	Nr_100		:BOOL;// #MText: #HText: #Prio: #BMK:
	Nr_101		:BOOL;// #MText: #HText: #Prio: #BMK:
	Nr_102		:BOOL;// #MText: #HText: #Prio: #BMK:
	Nr_103		:BOOL;// #MText: #HText: #Prio: #BMK:
	Nr_104		:BOOL;// #MText: #HText: #Prio: #BMK:
	Nr_105		:BOOL;// #MText: #HText: #Prio: #BMK:
	Nr_106		:BOOL;// #MText: #HText: #Prio: #BMK:
	Nr_107		:BOOL;// #MText: #HText: #Prio: #BMK:
	Nr_108		:BOOL;// #MText: #HText: #Prio: #BMK:
	Nr_109		:BOOL;// #MText: #HText: #Prio: #BMK:
	Nr_110		:BOOL;// #MText: #HText: #Prio: #BMK:
	Nr_111		:BOOL;// #MText: #HText: #Prio: #BMK:
	Nr_112		:BOOL;// #MText: #HText: #Prio: #BMK:
	Nr_113		:BOOL;// #MText: #HText: #Prio: #BMK:
	Nr_114		:BOOL;// #MText: #HText: #Prio: #BMK:
	Nr_115		:BOOL;// #MText: #HText: #Prio: #BMK:
	Nr_116		:BOOL;// #MText: #HText: #Prio: #BMK:
	Nr_117		:BOOL;// #MText: #HText: #Prio: #BMK:
	Nr_118		:BOOL;// #MText: #HText: #Prio: #BMK:
	Nr_119		:BOOL;// #MText: #HText: #Prio: #BMK:
	Nr_120		:BOOL;// #MText: #HText: #Prio: #BMK:
	Nr_121		:BOOL;// #MText: #HText: #Prio: #BMK:
	Nr_122		:BOOL;// #MText: #HText: #Prio: #BMK:
	Nr_123		:BOOL;// #MText: #HText: #Prio: #BMK:
	Nr_124		:BOOL;// #MText: #HText: #Prio: #BMK:
	Nr_125		:BOOL;// #MText: #HText: #Prio: #BMK:
	Nr_126		:BOOL;// #MText: #HText: #Prio: #BMK:
	Nr_127		:BOOL;// #MText: #HText: #Prio: #BMK:
	Nr_128		:BOOL;// #MText: #HText: #Prio: #BMK:
	Nr_129		:BOOL;// #MText: #HText: #Prio: #BMK:
	Nr_130		:BOOL;// #MText: #HText: #Prio: #BMK:
	Nr_131		:BOOL;// #MText: #HText: #Prio: #BMK:
	Nr_132		:BOOL;// #MText: #HText: #Prio: #BMK:
	Nr_133		:BOOL;// #MText: #HText: #Prio: #BMK:
	Nr_134		:BOOL;// #MText: #HText: #Prio: #BMK:
	Nr_135		:BOOL;// #MText: #HText: #Prio: #BMK:
	Nr_136		:BOOL;// #MText: #HText: #Prio: #BMK:
	Nr_137		:BOOL;// #MText: #HText: #Prio: #BMK:
	Nr_138		:BOOL;// #MText: #HText: #Prio: #BMK:
	Nr_139		:BOOL;// #MText: #HText: #Prio: #BMK:
	Nr_140		:BOOL;// #MText: #HText: #Prio: #BMK:
	Nr_141		:BOOL;// #MText: #HText: #Prio: #BMK:
	Nr_142		:BOOL;// #MText: #HText: #Prio: #BMK:
	Nr_143		:BOOL;// #MText: #HText: #Prio: #BMK:
	Nr_144		:BOOL;// #MText: #HText: #Prio: #BMK:
	Nr_145		:BOOL;// #MText: #HText: #Prio: #BMK:
	Nr_146		:BOOL;// #MText: #HText: #Prio: #BMK:
	Nr_147		:BOOL;// #MText: #HText: #Prio: #BMK:
	Nr_148		:BOOL;// #MText: #HText: #Prio: #BMK:
	Nr_149		:BOOL;// #MText: #HText: #Prio: #BMK:
	Nr_150		:BOOL;// #MText: #HText: #Prio: #BMK:
	Nr_151		:BOOL;// #MText: #HText: #Prio: #BMK:
	Nr_152		:BOOL;// #MText: #HText: #Prio: #BMK:
	Nr_153		:BOOL;// #MText: #HText: #Prio: #BMK:
	Nr_154		:BOOL;// #MText: #HText: #Prio: #BMK:
	Nr_155		:BOOL;// #MText: #HText: #Prio: #BMK:
	Nr_156		:BOOL;// #MText: #HText: #Prio: #BMK:
	Nr_157		:BOOL;// #MText: #HText: #Prio: #BMK:
	Nr_158		:BOOL;// #MText: #HText: #Prio: #BMK:
	Nr_159		:BOOL;// #MText: #HText: #Prio: #BMK:
	Nr_160		:BOOL;// #MText: #HText: #Prio: #BMK:
	Nr_161		:BOOL;// #MText: #HText: #Prio: #BMK:
	Nr_162		:BOOL;// #MText: #HText: #Prio: #BMK:
	Nr_163		:BOOL;// #MText: #HText: #Prio: #BMK:
	Nr_164		:BOOL;// #MText: #HText: #Prio: #BMK:
	Nr_165		:BOOL;// #MText: #HText: #Prio: #BMK:
	Nr_166		:BOOL;// #MText: #HText: #Prio: #BMK:
	Nr_167		:BOOL;// #MText: #HText: #Prio: #BMK:
	Nr_168		:BOOL;// #MText: #HText: #Prio: #BMK:
	Nr_169		:BOOL;// #MText: #HText: #Prio: #BMK:
	Nr_170		:BOOL;// #MText: #HText: #Prio: #BMK:
	Nr_171		:BOOL;// #MText: #HText: #Prio: #BMK:
	Nr_172		:BOOL;// #MText: #HText: #Prio: #BMK:
	Nr_173		:BOOL;// #MText: #HText: #Prio: #BMK:
	Nr_174		:BOOL;// #MText: #HText: #Prio: #BMK:
	Nr_175		:BOOL;// #MText: #HText: #Prio: #BMK:
	Nr_176		:BOOL;// #MText: #HText: #Prio: #BMK:
	Nr_177		:BOOL;// #MText: #HText: #Prio: #BMK:
	Nr_178		:BOOL;// #MText: #HText: #Prio: #BMK:
	Nr_179		:BOOL;// #MText: #HText: #Prio: #BMK:
	Nr_180		:BOOL;// #MText: #HText: #Prio: #BMK:
	Nr_181		:BOOL;// #MText: #HText: #Prio: #BMK:
	Nr_182		:BOOL;// #MText: #HText: #Prio: #BMK:
	Nr_183		:BOOL;// #MText: #HText: #Prio: #BMK:
	Nr_184		:BOOL;// #MText: #HText: #Prio: #BMK:
	Nr_185		:BOOL;// #MText: #HText: #Prio: #BMK:
	Nr_186		:BOOL;// #MText: #HText: #Prio: #BMK:
	Nr_187		:BOOL;// #MText: #HText: #Prio: #BMK:
	Nr_188		:BOOL;// #MText: #HText: #Prio: #BMK:
	Nr_189		:BOOL;// #MText: #HText: #Prio: #BMK:
	Nr_190		:BOOL;// #MText: #HText: #Prio: #BMK:
	Nr_191		:BOOL;// #MText: #HText: #Prio: #BMK:
	Nr_192		:BOOL;// #MText: #HText: #Prio: #BMK:
	Nr_193		:BOOL;// #MText: #HText: #Prio: #BMK:
	Nr_194		:BOOL;// #MText: #HText: #Prio: #BMK:
	Nr_195		:BOOL;// #MText: #HText: #Prio: #BMK:
	Nr_196		:BOOL;// #MText: #HText: #Prio: #BMK:
	Nr_197		:BOOL;// #MText: #HText: #Prio: #BMK:
	Nr_198		:BOOL;// #MText: #HText: #Prio: #BMK:
	Nr_199		:BOOL;// #MText: #HText: #Prio: #BMK:
	
END_STRUCT
END_TYPE

// ---- SRT_Allgemein/0010_Bausteine_mitDuts/DUTs/Meldungen/DUT_Meldungen_5000.TcDUT
TYPE DUT_Meldungen_5000 :
STRUCT
					  // #MText: Achtung ein Fehler #HText: Achtung eine Hilfe #Prio: 1-10 Error 11-20 Warnung 21-30 Info #BMK:	

	Nr_001		:BOOL;// #MText: #HText: #Prio: #BMK:
	Nr_002		:BOOL;// #MText: #HText: #Prio: #BMK: 
	Nr_003		:BOOL;// #MText: #HText: #Prio: #BMK: 
	Nr_004		:BOOL;// #MText: #HText: #Prio: #BMK: 
	Nr_005		:BOOL;// #MText: #HText: #Prio: #BMK: 
	Nr_006		:BOOL;// #MText: #HText: #Prio: #BMK: 
	Nr_007		:BOOL;// #MText: #HText: #Prio: #BMK: 
	Nr_008		:BOOL;// #MText: #HText: #Prio: #BMK: 
	Nr_009		:BOOL;// #MText: #HText: #Prio: #BMK: 
	Nr_010		:BOOL;// #MText: #HText: #Prio: #BMK: 
	Nr_011		:BOOL;// #MText: #HText: #Prio: #BMK: 
	Nr_012		:BOOL;// #MText: #HText: #Prio: #BMK: 
	Nr_013		:BOOL;// #MText: #HText: #Prio: #BMK: 
	Nr_014		:BOOL;// #MText: #HText: #Prio: #BMK: 
	Nr_015		:BOOL;// #MText: #HText: #Prio: #BMK:     
	Nr_016		:BOOL;// #MText: #HText: #Prio: #BMK:
	Nr_017		:BOOL;// #MText: #HText: #Prio: #BMK:     
	Nr_018		:BOOL;// #MText: #HText: #Prio: #BMK:
	Nr_019		:BOOL;// #MText: #HText: #Prio: #BMK:     
	Nr_020		:BOOL;// #MText: #HText: #Prio: #BMK:
	Nr_021		:BOOL;// #MText: #HText: #Prio: #BMK:     
	Nr_022		:BOOL;// #MText: #HText: #Prio: #BMK:     
	Nr_023		:BOOL;// #MText: #HText: #Prio: #BMK:      
	Nr_024		:BOOL;// #MText: #HText: #Prio: #BMK:
	Nr_025		:BOOL;// #MText: #HText: #Prio: #BMK:      
	Nr_026		:BOOL;// #MText: #HText: #Prio: #BMK:
	Nr_027		:BOOL;// #MText: #HText: #Prio: #BMK:      
	Nr_028		:BOOL;// #MText: #HText: #Prio: #BMK:
	Nr_029		:BOOL;// #MText: #HText: #Prio: #BMK:      
	Nr_030		:BOOL;// #MText: #HText: #Prio: #BMK:
	Nr_031		:BOOL;// #MText: #HText: #Prio: #BMK:      
	Nr_032		:BOOL;// #MText: #HText: #Prio: #BMK:
	Nr_033		:BOOL;// #MText: #HText: #Prio: #BMK:      
	Nr_034		:BOOL;// #MText: #HText: #Prio: #BMK:
	Nr_035		:BOOL;// #MText: #HText: #Prio: #BMK:      
	Nr_036		:BOOL;// #MText: #HText: #Prio: #BMK:
	Nr_037		:BOOL;// #MText: #HText: #Prio: #BMK:
	Nr_038		:BOOL;// #MText: #HText: #Prio: #BMK:
	Nr_039		:BOOL;// #MText: #HText: #Prio: #BMK:
	Nr_040		:BOOL;// #MText: #HText: #Prio: #BMK:
	Nr_041		:BOOL;// #MText: #HText: #Prio: #BMK:
	Nr_042		:BOOL;// #MText: #HText: #Prio: #BMK:
	Nr_043		:BOOL;// #MText: #HText: #Prio: #BMK:
	Nr_044		:BOOL;// #MText: #HText: #Prio: #BMK:
	Nr_045		:BOOL;// #MText: #HText: #Prio: #BMK:
	Nr_046		:BOOL;// #MText: #HText: #Prio: #BMK:
	Nr_047		:BOOL;// #MText: #HText: #Prio: #BMK:
	Nr_048		:BOOL;// #MText: #HText: #Prio: #BMK:
	Nr_049		:BOOL;// #MText: #HText: #Prio: #BMK:
	Nr_050		:BOOL;// #MText: #HText: #Prio: #BMK:
	Nr_051		:BOOL;// #MText: #HText: #Prio: #BMK:
	Nr_052		:BOOL;// #MText: #HText: #Prio: #BMK:
	Nr_053		:BOOL;// #MText: #HText: #Prio: #BMK:
	Nr_054		:BOOL;// #MText: #HText: #Prio: #BMK:
	Nr_055		:BOOL;// #MText: #HText: #Prio: #BMK:
	Nr_056		:BOOL;// #MText: #HText: #Prio: #BMK:
	Nr_057		:BOOL;// #MText: #HText: #Prio: #BMK:
	Nr_058		:BOOL;// #MText: #HText: #Prio: #BMK:
	Nr_059		:BOOL;// #MText: #HText: #Prio: #BMK:
	Nr_060		:BOOL;// #MText: #HText: #Prio: #BMK:
	Nr_061		:BOOL;// #MText: #HText: #Prio: #BMK:
	Nr_062		:BOOL;// #MText: #HText: #Prio: #BMK:
	Nr_063		:BOOL;// #MText: #HText: #Prio: #BMK:
	Nr_064		:BOOL;// #MText: #HText: #Prio: #BMK:
	Nr_065		:BOOL;// #MText: #HText: #Prio: #BMK:
	Nr_066		:BOOL;// #MText: #HText: #Prio: #BMK:
	Nr_067		:BOOL;// #MText: #HText: #Prio: #BMK:
	Nr_068		:BOOL;// #MText: #HText: #Prio: #BMK:
	Nr_069		:BOOL;// #MText: #HText: #Prio: #BMK:
	Nr_070		:BOOL;// #MText: #HText: #Prio: #BMK:
	Nr_071		:BOOL;// #MText: #HText: #Prio: #BMK:
	Nr_072		:BOOL;// #MText: #HText: #Prio: #BMK:
	Nr_073		:BOOL;// #MText: #HText: #Prio: #BMK:
	Nr_074		:BOOL;// #MText: #HText: #Prio: #BMK:
	Nr_075		:BOOL;// #MText: #HText: #Prio: #BMK:
	Nr_076		:BOOL;// #MText: #HText: #Prio: #BMK:
	Nr_077		:BOOL;// #MText: #HText: #Prio: #BMK:
	Nr_078		:BOOL;// #MText: #HText: #Prio: #BMK:
	Nr_079		:BOOL;// #MText: #HText: #Prio: #BMK:
	Nr_080		:BOOL;// #MText: #HText: #Prio: #BMK:
	Nr_081		:BOOL;// #MText: #HText: #Prio: #BMK:
	Nr_082		:BOOL;// #MText: #HText: #Prio: #BMK:
	Nr_083		:BOOL;// #MText: #HText: #Prio: #BMK:
	Nr_084		:BOOL;// #MText: #HText: #Prio: #BMK:
	Nr_085		:BOOL;// #MText: #HText: #Prio: #BMK:
	Nr_086		:BOOL;// #MText: #HText: #Prio: #BMK:
	Nr_087		:BOOL;// #MText: #HText: #Prio: #BMK:
	Nr_088		:BOOL;// #MText: #HText: #Prio: #BMK:
	Nr_089		:BOOL;// #MText: #HText: #Prio: #BMK:
	Nr_090		:BOOL;// #MText: #HText: #Prio: #BMK:
	Nr_091		:BOOL;// #MText: #HText: #Prio: #BMK:
	Nr_092		:BOOL;// #MText: #HText: #Prio: #BMK:
	Nr_093		:BOOL;// #MText: #HText: #Prio: #BMK:
	Nr_094		:BOOL;// #MText: #HText: #Prio: #BMK:
	Nr_095		:BOOL;// #MText: #HText: #Prio: #BMK:
	Nr_096		:BOOL;// #MText: #HText: #Prio: #BMK:
	Nr_097		:BOOL;// #MText: #HText: #Prio: #BMK:
	Nr_098		:BOOL;// #MText: #HText: #Prio: #BMK:
	Nr_099		:BOOL;// #MText: #HText: #Prio: #BMK:
	
	Nr_100		:BOOL;// #MText: #HText: #Prio: #BMK:
	Nr_101		:BOOL;// #MText: #HText: #Prio: #BMK:
	Nr_102		:BOOL;// #MText: #HText: #Prio: #BMK:
	Nr_103		:BOOL;// #MText: #HText: #Prio: #BMK:
	Nr_104		:BOOL;// #MText: #HText: #Prio: #BMK:
	Nr_105		:BOOL;// #MText: #HText: #Prio: #BMK:
	Nr_106		:BOOL;// #MText: #HText: #Prio: #BMK:
	Nr_107		:BOOL;// #MText: #HText: #Prio: #BMK:
	Nr_108		:BOOL;// #MText: #HText: #Prio: #BMK:
	Nr_109		:BOOL;// #MText: #HText: #Prio: #BMK:
	Nr_110		:BOOL;// #MText: #HText: #Prio: #BMK:
	Nr_111		:BOOL;// #MText: #HText: #Prio: #BMK:
	Nr_112		:BOOL;// #MText: #HText: #Prio: #BMK:
	Nr_113		:BOOL;// #MText: #HText: #Prio: #BMK:
	Nr_114		:BOOL;// #MText: #HText: #Prio: #BMK:
	Nr_115		:BOOL;// #MText: #HText: #Prio: #BMK:
	Nr_116		:BOOL;// #MText: #HText: #Prio: #BMK:
	Nr_117		:BOOL;// #MText: #HText: #Prio: #BMK:
	Nr_118		:BOOL;// #MText: #HText: #Prio: #BMK:
	Nr_119		:BOOL;// #MText: #HText: #Prio: #BMK:
	Nr_120		:BOOL;// #MText: #HText: #Prio: #BMK:
	Nr_121		:BOOL;// #MText: #HText: #Prio: #BMK:
	Nr_122		:BOOL;// #MText: #HText: #Prio: #BMK:
	Nr_123		:BOOL;// #MText: #HText: #Prio: #BMK:
	Nr_124		:BOOL;// #MText: #HText: #Prio: #BMK:
	Nr_125		:BOOL;// #MText: #HText: #Prio: #BMK:
	Nr_126		:BOOL;// #MText: #HText: #Prio: #BMK:
	Nr_127		:BOOL;// #MText: #HText: #Prio: #BMK:
	Nr_128		:BOOL;// #MText: #HText: #Prio: #BMK:
	Nr_129		:BOOL;// #MText: #HText: #Prio: #BMK:
	Nr_130		:BOOL;// #MText: #HText: #Prio: #BMK:
	Nr_131		:BOOL;// #MText: #HText: #Prio: #BMK:
	Nr_132		:BOOL;// #MText: #HText: #Prio: #BMK:
	Nr_133		:BOOL;// #MText: #HText: #Prio: #BMK:
	Nr_134		:BOOL;// #MText: #HText: #Prio: #BMK:
	Nr_135		:BOOL;// #MText: #HText: #Prio: #BMK:
	Nr_136		:BOOL;// #MText: #HText: #Prio: #BMK:
	Nr_137		:BOOL;// #MText: #HText: #Prio: #BMK:
	Nr_138		:BOOL;// #MText: #HText: #Prio: #BMK:
	Nr_139		:BOOL;// #MText: #HText: #Prio: #BMK:
	Nr_140		:BOOL;// #MText: #HText: #Prio: #BMK:
	Nr_141		:BOOL;// #MText: #HText: #Prio: #BMK:
	Nr_142		:BOOL;// #MText: #HText: #Prio: #BMK:
	Nr_143		:BOOL;// #MText: #HText: #Prio: #BMK:
	Nr_144		:BOOL;// #MText: #HText: #Prio: #BMK:
	Nr_145		:BOOL;// #MText: #HText: #Prio: #BMK:
	Nr_146		:BOOL;// #MText: #HText: #Prio: #BMK:
	Nr_147		:BOOL;// #MText: #HText: #Prio: #BMK:
	Nr_148		:BOOL;// #MText: #HText: #Prio: #BMK:
	Nr_149		:BOOL;// #MText: #HText: #Prio: #BMK:
	Nr_150		:BOOL;// #MText: #HText: #Prio: #BMK:
	Nr_151		:BOOL;// #MText: #HText: #Prio: #BMK:
	Nr_152		:BOOL;// #MText: #HText: #Prio: #BMK:
	Nr_153		:BOOL;// #MText: #HText: #Prio: #BMK:
	Nr_154		:BOOL;// #MText: #HText: #Prio: #BMK:
	Nr_155		:BOOL;// #MText: #HText: #Prio: #BMK:
	Nr_156		:BOOL;// #MText: #HText: #Prio: #BMK:
	Nr_157		:BOOL;// #MText: #HText: #Prio: #BMK:
	Nr_158		:BOOL;// #MText: #HText: #Prio: #BMK:
	Nr_159		:BOOL;// #MText: #HText: #Prio: #BMK:
	Nr_160		:BOOL;// #MText: #HText: #Prio: #BMK:
	Nr_161		:BOOL;// #MText: #HText: #Prio: #BMK:
	Nr_162		:BOOL;// #MText: #HText: #Prio: #BMK:
	Nr_163		:BOOL;// #MText: #HText: #Prio: #BMK:
	Nr_164		:BOOL;// #MText: #HText: #Prio: #BMK:
	Nr_165		:BOOL;// #MText: #HText: #Prio: #BMK:
	Nr_166		:BOOL;// #MText: #HText: #Prio: #BMK:
	Nr_167		:BOOL;// #MText: #HText: #Prio: #BMK:
	Nr_168		:BOOL;// #MText: #HText: #Prio: #BMK:
	Nr_169		:BOOL;// #MText: #HText: #Prio: #BMK:
	Nr_170		:BOOL;// #MText: #HText: #Prio: #BMK:
	Nr_171		:BOOL;// #MText: #HText: #Prio: #BMK:
	Nr_172		:BOOL;// #MText: #HText: #Prio: #BMK:
	Nr_173		:BOOL;// #MText: #HText: #Prio: #BMK:
	Nr_174		:BOOL;// #MText: #HText: #Prio: #BMK:
	Nr_175		:BOOL;// #MText: #HText: #Prio: #BMK:
	Nr_176		:BOOL;// #MText: #HText: #Prio: #BMK:
	Nr_177		:BOOL;// #MText: #HText: #Prio: #BMK:
	Nr_178		:BOOL;// #MText: #HText: #Prio: #BMK:
	Nr_179		:BOOL;// #MText: #HText: #Prio: #BMK:
	Nr_180		:BOOL;// #MText: #HText: #Prio: #BMK:
	Nr_181		:BOOL;// #MText: #HText: #Prio: #BMK:
	Nr_182		:BOOL;// #MText: #HText: #Prio: #BMK:
	Nr_183		:BOOL;// #MText: #HText: #Prio: #BMK:
	Nr_184		:BOOL;// #MText: #HText: #Prio: #BMK:
	Nr_185		:BOOL;// #MText: #HText: #Prio: #BMK:
	Nr_186		:BOOL;// #MText: #HText: #Prio: #BMK:
	Nr_187		:BOOL;// #MText: #HText: #Prio: #BMK:
	Nr_188		:BOOL;// #MText: #HText: #Prio: #BMK:
	Nr_189		:BOOL;// #MText: #HText: #Prio: #BMK:
	Nr_190		:BOOL;// #MText: #HText: #Prio: #BMK:
	Nr_191		:BOOL;// #MText: #HText: #Prio: #BMK:
	Nr_192		:BOOL;// #MText: #HText: #Prio: #BMK:
	Nr_193		:BOOL;// #MText: #HText: #Prio: #BMK:
	Nr_194		:BOOL;// #MText: #HText: #Prio: #BMK:
	Nr_195		:BOOL;// #MText: #HText: #Prio: #BMK:
	Nr_196		:BOOL;// #MText: #HText: #Prio: #BMK:
	Nr_197		:BOOL;// #MText: #HText: #Prio: #BMK:
	Nr_198		:BOOL;// #MText: #HText: #Prio: #BMK:
	Nr_199		:BOOL;// #MText: #HText: #Prio: #BMK:
	
END_STRUCT
END_TYPE

// ---- SRT_Allgemein/0010_Bausteine_mitDuts/DUTs/Rexroth FU/DUT_Rexroth_FU_steuern.TcDUT
TYPE DUT_Rexroth_FU_steuern :
STRUCT
	vor					:BOOL;
	zur					:BOOL;
	rampe				:INT;
	speed				:REAL;
	speed_hand			:REAL;   
	reglerfreigabe		:BOOL;
END_STRUCT
END_TYPE

// ---- SRT_Allgemein/0010_Bausteine_mitDuts/DUTs/Safety/ST_InfoDataConnection_1918.TcDUT
TYPE ST_InfoDataConnection_1918 :
STRUCT
	usiMapState		: USINT;
	usiMapDiag		: USINT;
	bSignals_1		: BIT;
	bSignals_1_fault: BIT;
	bSignals_2		: BIT;
	bSignals_2_fault: BIT;
	bSignals_3		: BIT;
	bSignals_3_fault: BIT;
	bSignals_4		: BIT;
	bSignals_4_fault: BIT;
	bSignals_5		: BIT;
	bSignals_5_fault: BIT;
	bSignals_6		: BIT;
	bSignals_6_fault: BIT;
	bSignals_7		: BIT;
	bSignals_7_fault: BIT;
	bSignals_8		: BIT;
	bSignals_8_fault: BIT;
END_STRUCT
END_TYPE

// ---- SRT_Allgemein/0010_Bausteine_mitDuts/DUTs/Servo/DUT_Achse_Service.TcDUT
TYPE DUT_Achse_Service :
STRUCT

   betriebsart 			: INT ;		(*	Betriebsarten:1=Tippen,2=Position1,4=Referenzieren *)
   plus_start 			: BOOL; 	(*	Tippen plus / Start positionierung *)
   minus_stop 			: BOOL ;	(*	Tippen minus / Stopp positionierung *)
   override 			: INT ;		(*	Geschwindigkeit in % *)
   sollpos_hand 		: REAL ;	(*	Position 1 *)
   pos_2 				: REAL ;	(*	Position 2 *)
   zeit 				: INT ;		(*	Verweilzeit *)
   istpos 				: REAL ;	(*	Istposition *)
   status				: DWORD ;

END_STRUCT
END_TYPE

// ---- SRT_Allgemein/0010_Bausteine_mitDuts/DUTs/Servo/DUT_Achse_Status.TcDUT
TYPE DUT_Achse_Status :
STRUCT
	ist_pos				: REAL;				(*  aktuelle ist Position  *)                          
	in_pos				: BOOL;				(*  Achse in Position (Soll=IST + - Positionsfenster) *)
	ziel_pos			: REAL;				(*  Aktuelle Zielposition der Achse *)
	nicht_ref			: BOOL;				(*  Achse ist nicht referenziert  *)                  
    bremse				: BOOL;				(*  Bremse lösen *)                                     
	Achs_Status			: ST_AxisStatus;	(* 	aktueller Achsstatus *)
	Drehmoment_aktiv	: BOOL;				(*	Betriebsart Drehmoment aktiv	*)                   
	Drehmoment_erreicht	: BOOL;				(*	Drehmoment erreicht	*)        
	Bremsentest_notwendig	: BOOL;            
END_STRUCT
END_TYPE

// ---- SRT_Allgemein/0010_Bausteine_mitDuts/DUTs/Servo/DUT_PD_InOut_Achsen.TcDUT
TYPE DUT_PD_InOut_Achsen :
STRUCT
	S0145_steuerword			AT%Q*:WORD;		// Signal Steuerwort für den Bremsentest/Reset des Umrichters
												// 	.0 = Reset, 				S-0-0099 - C0500 Reset Zustandsklasse 1
												//	.1 = Absolutwert setzen, 	S-0-0447 - C0300 Absolutwert setzen   !!! nur ohne Reglerfreigabe möglich
												//	.2 = Bremsentest, 			P-0-0541 - C2100 Kommando Haltesystemüberwachen 
	S0052_ref_pos				AT%Q*:DINT;		// Referenzposition /Absolutwert zum setzen
	S0092_drehmoment_grenzwert 	AT%Q*:UINT;		// Drehmoment/ Kraft Grenzwert bipolar


	S0144_statusword			AT%I*:WORD;		// Signal Statuswort 
	P0539_status_bremse			AT%I*:WORD;		// Signal Statuswort für den Bremsentest
	S0390_diagnose				AT%I*:DWORD;	// Diagnose Word des Reglers

	//***** Nur beim Achsmodul XMD *********************************************************************
	P0115_axis_state_maschine	AT%I*:WORD;		//	Achs-State-Machine: Statuswort, Achse 
												//	.0 -> 1=Der Wechselrichter erlaubt die Leistungsfreigabe
	S0240_DCbus_Supply			AT%Q*:WORD;		//	Zwischenkreis-Versorgung: Steuerwort										
												//	.0-> 1=der Zwischenkreis ist bereit zur Leistungsabgabe		
										
	//***** Nur beim Versorgungsmodul XCS **************************************************************
	S2058_power_supply_status	AT%I*:WORD;		// Zwischenkreis-Versorgung: Steuerwort		
												//	.15-> 1= Die Freigabe ist gegeben, d.h. der Zwischenkreis ist belastbar
	S2057_power_supply_contol	AT%Q*:WORD;		//	Versorgerregelung: Steuerwort 
												//	.12-> 1= Kontakt schließen, Freigabe
												//	.14-> 1= Zwischenkreis laden
												//	.15-> 1= Freigabe, Sollbetriebsart aktivieren
END_STRUCT
END_TYPE

// ---- SRT_Allgemein/0010_Bausteine_mitDuts/DUTs/Servo/DUT_Rexroth_Parameter.TcDUT
TYPE DUT_Rexroth_Parameter :
STRUCT
	Beschleunigung	:LREAL;
	Verzoegerung	:LREAL;
	Ruck			:LREAL;
END_STRUCT
END_TYPE

// ---- SRT_Allgemein/0010_Bausteine_mitDuts/DUTs/SEW_Movitrac/COE/st_COE_Parameter.TcDUT
TYPE st_COE_Parameter :
STRUCT
	sName		: STRING(22);
	nSubIndex 	 : BYTE;
   	nIndex   		 : WORD;
	nWert		: DWORD;
	nLength		: UDINT;
	nZugriff		: BYTE:= 0;	(* 0 = lesen| 1 = schreiben | 2 = lesen und schreiben | 3 = ende *)
	nFaktor		: LREAL	:=	1;
END_STRUCT
END_TYPE

// ---- SRT_Allgemein/0010_Bausteine_mitDuts/DUTs/SEW_Movitrac/DUT_SEW_FU_Status.TcDUT
TYPE DUT_SEW_FU_Status :
STRUCT

	nicht_bereit		:BOOL;	(* Umrichter ist nicht betriebsbereit *)
	ist_drehzahl		:REAL;	(* aktuelle Drehzahl *)
	ist_drehzahl_90		:BOOL;	(* 90% der Soll Drehzahl erreicht *)
	antriebAktiv		:BOOL;	(* Dreht mehr als 1 rpm*)
	ist_strom			:REAL;	(* aktueller Strom *)
	ist_drehmoment		:REAL;	(* aktuelles Drehmoment *)
END_STRUCT
END_TYPE

// ---- SRT_Allgemein/0010_Bausteine_mitDuts/DUTs/SEW_Movitrac/DUT_SEW_FU_Visu.TcDUT
TYPE DUT_SEW_FU_Visu :
STRUCT
	plus_start			:BOOL;	(* Motor ein *)
	minus_stop			:BOOL;	(* Motor aus *)
	betriebsart			:INT;	(* 0=keine , 1=Tippen, 2=Vorwärts, 3=Rückwärts 4=Option 5= CoE-Daten*)
	override			:REAL;	(* Anlagenoverride *)
	istdrehzahl			:REAL;	(* Ist-Drehzahl *)
	iststrom			:REAL;
	diagnose			:INT;	(* Status und Fehlerverweis auf die Diagnoseliste*)
	status				:INT;	(* Buttonstatus (Farbzuweisung)*)
	Para				:DUT_SEW_Para;
END_STRUCT
END_TYPE

// ---- SRT_Allgemein/0010_Bausteine_mitDuts/DUTs/Ventil/DUT_Ventil_para.TcDUT
TYPE DUT_Ventil_para :
STRUCT
	ueberwachung_vor_aktiv	:BOOL:=TRUE;	//0 = Endlagenüberwachung vor deaktiviert
	ueberwachung_zur_aktiv	:BOOL:=TRUE;	//0 = Endlagenüberwachung zurück deaktiviert
	ausgang_vor_halten		:BOOL:=FALSE;	//1 = Ausgang immer Ein, sonst 0 in Endlage/1 nicht in Endlage
	ausgang_zur_halten		:BOOL:=FALSE;	//1 = Ausgang immer Ein, sonst 0 in Endlage/1 nicht in Endlage
	entprellen_vor_aktiv	:BOOL:=TRUE;	//0 = Endlage sofort überwachen wenn einmal erreicht
	entprellen_zur_aktiv	:BOOL:=TRUE;	//0 = Endlage sofort überwachen wenn einmal erreicht
	ueberwachungszeit_vor	:TIME:=T#10S;	//Überwachungszeit in ms (0-30000ms)
	ueberwachungszeit_zur	:TIME:=T#10S;	//Überwachungszeit in ms (0-30000ms)
	entprellungszeit_vor	:TIME:=T#50MS;	//Entprellungszeit in ms (0-10000ms)
	entprellungszeit_zur	:TIME:=T#50MS;	//Entprellungszeit in ms (0-10000ms)
END_STRUCT
END_TYPE

// ---- SRT_Allgemein/0010_Bausteine_mitDuts/DUTs/Ventil/DUT_Ventil_VISU.TcDUT
TYPE DUT_Ventil_VISU :
STRUCT
	hand_vor				:BOOL;	//Hand vorfahren
	hand_zur				:BOOL;	//Hand zurückfahren
	reset					:BOOL;	//intern gespeicherte Startsignale löschen
	service					:BOOL;	//1 = ALLE Überwachungen deaktiviert
	status					:BYTE;	//0=??? 1=vor 2=ist vor 3=fehler vor 4=zur 5=ist zur 6=Fehler zur 7=Fehler vor zur
	para					:DUT_Ventil_para;
END_STRUCT
END_TYPE

// ---- SRT_Allgemein/Bus/DUT_Busdiagnose.TcDUT
TYPE DUT_Busdiagnose :
STRUCT
	AmsNetId AT%I* :T_AmsNetIdArr;
		
	AnzahlTeilnehmer:UINT;//Busdiagnose - Tatsächliche Anzahl der teilnehmer
	FehlerfreiAktiv:BOOL; //Busdiagnose - Start für Visu
	Update:UINT; //Busdiagnose - Trigger für Visu
	AnzahlFehler:UINT; //Busdiagnose - Anzahl gestörter teilnehmer
	Daten:ARRAY [0..300] OF DUT_Busdiagnose_Daten; //Busdiagnose - Daten für Visu
END_STRUCT
END_TYPE

// ---- 0000/GVL_Visu_0000.TcGVL

VAR_GLOBAL
    KommAnVisu                 	: INT;      (* Kommunikation an die Visualisierung *)
    KommVonVisu                	: INT;      (* Kommunikation von der Visualisierung *)
    belegt                     	: BOOL;     (* true = erzeugt Dummyteil, false = keine Auswirkungen (nur Handauflage) *)
    daten_gebucht              	: BOOL;
    SteuerStatus              	: DUT_Visu_SteuerStatus;
	quittieren					: BOOL;
	override 					: INT;
    // Frequenzumrichter
    //transport                : DUT_SEW_FU_Visu;       //#Tab:  #Name: 

    // Servoregler
    //Achse                    : DUT_Achse_Service;      //#Tab: #Name: 

    // Ventile
    //Ventil                   : DUT_Ventil_VISU;        //#Tab: #Name: 

END_VAR

VAR_GLOBAL PERSISTENT
    Schrittnummer              : INT;
    //Kopfdaten                : DUT_Kopfdaten;
    //Kopfdaten_default        : DUT_Kopfdaten;
    //Jobdaten                 : DUT_Jobdaten;
    //Jobdaten_default         : DUT_Jobdaten;

    //para_Vorlage             : REAL := 0.0; //#Typ: VParam #Tab:  #Name:  #Einheit:mm #Min: 1 #Max: 100 #Format:F1
END_VAR

// ---- 1000_Allgemein/EAs_1000.TcGVL

{attribute 'linkalways'} 
VAR_GLOBAL

    // Eingaenge
    //_______________________________________________________

    // +FS1-3K5

        {attribute 'TcLinkTo' := 'TIID^Device 1 (EtherCAT)^+FS1-3K1 (BK1120)^+FS1-3K5 (EL1809)^Channel 5^Input'}
        e_FR_1000_Allgemein_Druckluft_OK AT %I* : BOOL; (* =FR.1000 Allgemein Druckluft OK *)
END_VAR

// ---- 1000_Allgemein/GVL_1000.TcGVL

VAR_GLOBAL
    // Achsen ***************************************************
    //Achse_steuern                     : DUT_Achse_Steuern;
    //Achse_status                      : DUT_Achse_Status;

    // Frequenzumrichter ****************************************
    //transport_steuern                 : DUT_SEW_FU_Steuern;
    //transport_status                  : DUT_SEW_FU_Status;

    // Ventile **************************************************
    //Ventil                            : DUT_Ventil_sps;

    // interne Variablen ****************************************
    sk_Freigabe                         : BOOL;
    sk                                  : INT;
    transport_einfoerdern_bereit        : BOOL;
    transport_ausfoerdern_bereit        : BOOL;

    Tuer_Anwahl                         : BOOL;   // Signal Tür Anwahl, Tür soll geöffnet werden
    Tuer_Freigabe                       : BOOL;   // Signal Tür Freigabe, Tür kann geöffnet werden
	
	
	Master_AmsNetId						:T_AmsNetID	:='172.16.1.000.1.1';		// Net id des EC- Masters
	TC_AmsNetId							:T_AmsNetID :='172.16.1.227.1.1';      	//	Net id des TwincatSystems
END_VAR
    

{attribute 'qualified_only'}
VAR_GLOBAL CONSTANT
	MaxCOEParam							:INT := 92;
	MAX_CSV_BASE_ROWS 					:INT := 92;
	iMaxEC								:INT := 0;								// Anzahl der verbauten EtherCat Klemmen
	MaxECDevices						:INT := 0;
	                                    
	ibn0								: BOOL;									// Am Ende müssen alle QUerverweise gelöscht werden
	ibn1								: BOOL := TRUE;							// Am Ende müssen alle QUerverweise gelöscht werden
		
END_VAR

// ---- 1000_Allgemein/GVL_Visu_1000.TcGVL

VAR_GLOBAL
    KommAnVisu                 : INT;      (* Kommunikation an die Visualisierung *)
    KommVonVisu                : INT;      (* Kommunikation von der Visualisierung *)
    belegt                     : BOOL;     (* true = erzeugt Dummyteil, false = keine Auswirkungen (nur Handauflage) *)
    daten_gebucht              : BOOL;
    SteuerStatus               : DUT_Visu_SteuerStatus;

    // Frequenzumrichter
    //transport                : DUT_SEW_FU_Visu;       //#Tab:  #Name: 

    // Servoregler
    //Achse                    : DUT_Achse_Service;      //#Tab: #Name: 

    // Ventile
    //Ventil                   : DUT_Ventil_VISU;        //#Tab: #Name: 

END_VAR

VAR_GLOBAL PERSISTENT
    Schrittnummer              : INT;
    //Kopfdaten                : DUT_Kopfdaten;
    //Kopfdaten_default        : DUT_Kopfdaten;
    //Jobdaten                 : DUT_Jobdaten;
    //Jobdaten_default         : DUT_Jobdaten;

    //para_Vorlage             : REAL := 0.0; //#Typ: VParam #Tab:  #Name:  #Einheit:mm #Min: 1 #Max: 100 #Format:F1
END_VAR

// ---- 3100_Bohraggregat/GVL_Visu_3100.TcGVL

VAR_GLOBAL
    KommAnVisu                 : INT;      (* Kommunikation an die Visualisierung *)
    KommVonVisu                : INT;      (* Kommunikation von der Visualisierung *)
    belegt                     : BOOL;     (* true = erzeugt Dummyteil, false = keine Auswirkungen (nur Handauflage) *)
    daten_gebucht              : BOOL;
    SteuerStatus               : DUT_Visu_SteuerStatus;

    // Frequenzumrichter
	Bohraggr_Schlosskast		: DUT_SEW_FU_Visu; 		//#Tab: 3100 Bohraggregat #Name: Bohraggregat Schlosskasten
	Bohraggr_Vorbohren			: DUT_SEW_FU_Visu; 		//#Tab: 3100 Bohraggregat #Name: Bohraggregat Vorbohren
	Bohraggr_Stulpfraes			: DUT_SEW_FU_Visu; 		//#Tab: 3100 Bohraggregat #Name: Bohraggregat Stulpfräser

    // Servoregler
	X_Achse						: DUT_Achse_Service;	//#Tab: 3100 Bohraggregat #Name: X-Achse 
	Y_Achse						: DUT_Achse_Service;	//#Tab: 3100 Bohraggregat #Name: Y-Achse 
	Z_Achse						: DUT_Achse_Service;	//#Tab: 3100 Bohraggregat #Name: Z-Achse 

    // Ventile
     Schlosskast_Vorlegehub            			: DUT_Ventil_VISU;        //#Tab: 3100 Bohraggregat #Name: Schlosskasten Vorlegehub
	 Vorbohren_Bohrhub        					: DUT_Ventil_VISU;        //#Tab: 3100 Bohraggregat #Name: Vorbohren Bohrhub
     Stulpfraes_Vorlegehub 						: DUT_Ventil_VISU;        //#Tab: 3100 Bohraggregat #Name: Stulpfräser Vorlegehub
     Nullkante 									: DUT_Ventil_VISU;        //#Tab: 3100 Bohraggregat #Name: Nullkante
     Schienenklemm								: DUT_Ventil_VISU;        //#Tab: 3100 Bohraggregat #Name: Schienenklemmung

END_VAR

VAR_GLOBAL PERSISTENT
    Schrittnummer              : INT;
    //Kopfdaten                : DUT_Kopfdaten;
    //Kopfdaten_default        : DUT_Kopfdaten;
    //Jobdaten                 : DUT_Jobdaten;
    //Jobdaten_default         : DUT_Jobdaten;

    //para_Vorlage             : REAL := 0.0; //#Typ: VParam #Tab:  #Name:  #Einheit:mm #Min: 1 #Max: 100 #Format:F1
END_VAR

// ---- 3200_Bohraggregat/GVL_3200.TcGVL

VAR_GLOBAL
    // Achsen ***************************************************	
	X_Achse_steuern						: DUT_Achse_Steuern;	
	X_Achse_status						: DUT_Achse_Status;	
		                            	
	Y_Achse_steuern						: DUT_Achse_Steuern;		
	Y_Achse_status						: DUT_Achse_Status;		
	
	Z_Achse_steuern						: DUT_Achse_Steuern;			
	Z_Achse_status						: DUT_Achse_Status;		

    // Frequenzumrichter ****************************************
	Bohraggr_Stufenbohr_steuern			: DUT_SEW_FU_Steuern;	
	Bohraggr_Stufenbohr_status			: DUT_SEW_FU_Status;
	Bohraggr_Stulpfraes_steuern			: DUT_SEW_FU_Steuern;	
	Bohraggr_Stulpfraes_status			: DUT_SEW_FU_Status;

    // Ventile **************************************************
    Vorbohren_Bohrhub          			: DUT_Ventil_sps;
    Stulpfraes_Vorlegehub      			: DUT_Ventil_sps;
    Pusher				             	: DUT_Ventil_sps;
    Schienenklemm		             	: DUT_Ventil_sps;

    // interne Variablen ****************************************
    sk_Freigabe                         : BOOL;
    sk                                  : INT;
    transport_einfoerdern_bereit        : BOOL;
    transport_ausfoerdern_bereit        : BOOL;

    Tuer_Anwahl                         : BOOL;   // Signal Tür Anwahl, Tür soll geöffnet werden
    Tuer_Freigabe                       : BOOL;   // Signal Tür Freigabe, Tür kann geöffnet werden
END_VAR

// ---- 3200_Bohraggregat/GVL_Visu_3200.TcGVL

VAR_GLOBAL
    KommAnVisu                 : INT;      (* Kommunikation an die Visualisierung *)
    KommVonVisu                : INT;      (* Kommunikation von der Visualisierung *)
    belegt                     : BOOL;     (* true = erzeugt Dummyteil, false = keine Auswirkungen (nur Handauflage) *)
    daten_gebucht              : BOOL;
    SteuerStatus               : DUT_Visu_SteuerStatus;

    // Frequenzumrichter
	Bohraggr_Stufenbohr			: DUT_SEW_FU_Visu; 		//#Tab: 3200 Bohraggregat #Name: Bohraggregat Stufenbohrer
	Bohraggr_Stulpfraes			: DUT_SEW_FU_Visu; 		//#Tab: 3200 Bohraggregat #Name: Bohraggregat Stulpfräser

    // Servoregler
	X_Achse						: DUT_Achse_Service;	//#Tab: 3200 Bohraggregat #Name: X-Achse 
	Y_Achse						: DUT_Achse_Service;	//#Tab: 3200 Bohraggregat #Name: Y-Achse 
	Z_Achse						: DUT_Achse_Service;	//#Tab: 3200 Bohraggregat #Name: Z-Achse 

    // Ventile
	 Vorbohren_Bohrhub        	: DUT_Ventil_VISU;        //#Tab: 3200 Bohraggregat #Name: Vorbohren Bohrhub
     Stulpfraes_Vorlegehub 		: DUT_Ventil_VISU;        //#Tab: 3200 Bohraggregat #Name: Stulpfräser Vorlegehub
     Pusher						: DUT_Ventil_VISU;        //#Tab: 3200 Bohraggregat #Name: Pusher 
     Schienenklemm				: DUT_Ventil_VISU;        //#Tab: 3200 Bohraggregat #Name: Schienenklemmung

END_VAR

VAR_GLOBAL PERSISTENT
    Schrittnummer              : INT;
    //Kopfdaten                : DUT_Kopfdaten;
    //Kopfdaten_default        : DUT_Kopfdaten;
    //Jobdaten                 : DUT_Jobdaten;
    //Jobdaten_default         : DUT_Jobdaten;

    //para_Vorlage             : REAL := 0.0; //#Typ: VParam #Tab:  #Name:  #Einheit:mm #Min: 1 #Max: 100 #Format:F1
END_VAR

// ---- 3300_Bohraggregat/EAs_3300.TcGVL
{attribute 'qualified_only'}
{attribute 'linkalways'} 
VAR_GLOBAL

	// Servoregler *************************************************************************************************************************************************

	{attribute 'TcNcAxis':='=3300+FS2-11M1 (X-Achse)'}	
	ea_X_Achse					: Axis_ref;				// Schnittstellen Struktur zwischen NC<->SPS
	
	{attribute 'TcNcAxis':='=3300+FS2-12M1 (Y-Achse)'}	
	ea_Y_Achse					: Axis_ref;				// Schnittstellen Struktur zwischen NC<->SPS

    // Umrichter
    //_______________________________________________________

	 {attribute 'TcLinkTo' := '	.PD_1_STATUSWORT  		:= TIID^Device 1 (EtherCAT)^=3300+FS2-16T1 (Bohraggr Schlüsselloch unten)^Module 1 (Standard 16 PD)^Inputs 16 PD^PI 1;
								.PD_2_IST_DREHZAHL  	:= TIID^Device 1 (EtherCAT)^=3300+FS2-16T1 (Bohraggr Schlüsselloch unten)^Module 1 (Standard 16 PD)^Inputs 16 PD^PI 2;
								.PD_3_Status  			:= TIID^Device 1 (EtherCAT)^=3300+FS2-16T1 (Bohraggr Schlüsselloch unten)^Module 1 (Standard 16 PD)^Inputs 16 PD^PI 3;
								.PD_4_IST_DREHMOMENT  	:= TIID^Device 1 (EtherCAT)^=3300+FS2-16T1 (Bohraggr Schlüsselloch unten)^Module 1 (Standard 16 PD)^Inputs 16 PD^PI 4;
								.PD_5_IST_STROM  		:= TIID^Device 1 (EtherCAT)^=3300+FS2-16T1 (Bohraggr Schlüsselloch unten)^Module 1 (Standard 16 PD)^Inputs 16 PD^PI 5'}		
		e_Bohraggr_Schluessel_un AT%I*	: DUT_SEW_FU_PD_IN; 	// Schnittstelle zwischen SPS und FU
	 {attribute 'TcLinkTo' := '	.PD_1_Steuerwort  		:= TIID^Device 1 (EtherCAT)^=3300+FS2-16T1 (Bohraggr Schlüsselloch unten)^Module 1 (Standard 16 PD)^Outputs 16 PD^PO 1;
								.PD_2_Solldrehzahl  	:= TIID^Device 1 (EtherCAT)^=3300+FS2-16T1 (Bohraggr Schlüsselloch unten)^Module 1 (Standard 16 PD)^Outputs 16 PD^PO 2;
								.PD_3_Sollbeschleunigung:= TIID^Device 1 (EtherCAT)^=3300+FS2-16T1 (Bohraggr Schlüsselloch unten)^Module 1 (Standard 16 PD)^Outputs 16 PD^PO 3;
								.PD_4_Sollverzoegerung  := TIID^Device 1 (EtherCAT)^=3300+FS2-16T1 (Bohraggr Schlüsselloch unten)^Module 1 (Standard 16 PD)^Outputs 16 PD^PO 4;
								.PD_5_Digitalausgaenge  := TIID^Device 1 (EtherCAT)^=3300+FS2-16T1 (Bohraggr Schlüsselloch unten)^Module 1 (Standard 16 PD)^Outputs 16 PD^PO 5'}
		a_Bohraggr_Schluessel_un AT%Q*	: DUT_SEW_FU_PD_OUT;	// Schnittstelle zwischen SPS und FU


    // Eingaenge
    //_______________________________________________________

    // +FS1-3K5

        {attribute 'TcLinkTo' := 'TIID^Device 1 (EtherCAT)^+FS1-3K1 (BK1120)^+FS1-3K5 (EL1809)^Channel 11^Input'}
        e_FR_3300_Bohraggregat_6_Schluesselloch_unten_Stillstandserkennung_Motor_steht AT %I* : BOOL; (* =FR.3300 Bohraggregat 6 (Schlüsselloch unten) Stillstandserkennung Motor steht *)

    // +K110-1K2

        {attribute 'TcLinkTo' := 'TIID^Device 1 (EtherCAT)^+K110-1K1 (BK1120)^+K110-1K2 (EL1809)^Channel 12^Input'}
        e_FR_3300_Druecker_Schluesselloch_unten_Bohraggregat_6_Bohrhub_ist_oben AT %I* : BOOL; (* =FR.3300 Drücker/Schlüsselloch unten Bohraggregat 6 Bohrhub ist oben *)

        {attribute 'TcLinkTo' := 'TIID^Device 1 (EtherCAT)^+K110-1K1 (BK1120)^+K110-1K2 (EL1809)^Channel 13^Input'}
        e_FR_3300_Druecker_Schluesselloch_unten_Bohraggregat_6_Bohrhub_ist_unten AT %I* : BOOL; (* =FR.3300 Drücker/Schlüsselloch unten Bohraggregat 6 Bohrhub ist unten *)


    // Ausgaenge
    //_______________________________________________________

    // +K110-2K1

        {attribute 'TcLinkTo' := 'TIID^Device 1 (EtherCAT)^+K110-1K1 (BK1120)^+K110-2K1 (EL2809)^Channel 13^Output'}
        a_FR_3300_Druecker_Schluesselloch_unten_Bohraggregat_6_Bohrhub_heben AT %Q* : BOOL; (* =FR.3300 Drücker/Schlüsselloch unten Bohraggregat 6 Bohrhub heben *)

        {attribute 'TcLinkTo' := 'TIID^Device 1 (EtherCAT)^+K110-1K1 (BK1120)^+K110-2K1 (EL2809)^Channel 14^Output'}
        a_FR_3300_Druecker_Schluesselloch_unten_Bohraggregat_6_Bohrhub_senken AT %Q* : BOOL; (* =FR.3300 Drücker/Schlüsselloch unten Bohraggregat 6 Bohrhub senken *)
END_VAR

// ---- 3300_Bohraggregat/GVL_Visu_3300.TcGVL

VAR_GLOBAL
    KommAnVisu                 : INT;      (* Kommunikation an die Visualisierung *)
    KommVonVisu                : INT;      (* Kommunikation von der Visualisierung *)
    belegt                     : BOOL;     (* true = erzeugt Dummyteil, false = keine Auswirkungen (nur Handauflage) *)
    daten_gebucht              : BOOL;
    SteuerStatus               : DUT_Visu_SteuerStatus;

    // Frequenzumrichter
	Bohraggr_Schluessel_un		: DUT_SEW_FU_Visu; 		//#Tab: 3300 Bohraggregat #Name: Bohraggregat Schlüsselkasten unten

    // Servoregler
	X_Achse						: DUT_Achse_Service;	//#Tab: 3300 Bohraggregat #Name: X-Achse 
	Y_Achse						: DUT_Achse_Service;	//#Tab: 3300 Bohraggregat #Name: Y-Achse 

    // Ventile
	 Schluessel_un_Bohrhub       : DUT_Ventil_VISU;     //#Tab: 3300 Bohraggregat #Name: Schlüsselkasten unten Bohrhub 

END_VAR

VAR_GLOBAL PERSISTENT
    Schrittnummer              : INT;
    //Kopfdaten                : DUT_Kopfdaten;
    //Kopfdaten_default        : DUT_Kopfdaten;
    //Jobdaten                 : DUT_Jobdaten;
    //Jobdaten_default         : DUT_Jobdaten;

    //para_Vorlage             : REAL := 0.0; //#Typ: VParam #Tab:  #Name:  #Einheit:mm #Min: 1 #Max: 100 #Format:F1
END_VAR

// ---- 3400_Bohraggregat/EAs_3400.TcGVL
{attribute 'qualified_only'}
{attribute 'linkalways'} 
VAR_GLOBAL

	// Servoregler *************************************************************************************************************************************************

	{attribute 'TcNcAxis':='=3400+FS2-11M1 (X-Achse)'}	
	ea_X_Achse					: Axis_ref;				// Schnittstellen Struktur zwischen NC<->SPS
	
	{attribute 'TcNcAxis':='=3400+FS2-12M1 (Y-Achse)'}	
	ea_Y_Achse					: Axis_ref;				// Schnittstellen Struktur zwischen NC<->SPS

    // Umrichter
    //_______________________________________________________
	
	 {attribute 'TcLinkTo' := '	.PD_1_STATUSWORT  		:= TIID^Device 1 (EtherCAT)^=3400+FS2-16T1 (Bohraggr Schlüsselloch oben)^Module 1 (Standard 16 PD)^Inputs 16 PD^PI 1;
								.PD_2_IST_DREHZAHL  	:= TIID^Device 1 (EtherCAT)^=3400+FS2-16T1 (Bohraggr Schlüsselloch oben)^Module 1 (Standard 16 PD)^Inputs 16 PD^PI 2;
								.PD_3_Status  			:= TIID^Device 1 (EtherCAT)^=3400+FS2-16T1 (Bohraggr Schlüsselloch oben)^Module 1 (Standard 16 PD)^Inputs 16 PD^PI 3;
								.PD_4_IST_DREHMOMENT  	:= TIID^Device 1 (EtherCAT)^=3400+FS2-16T1 (Bohraggr Schlüsselloch oben)^Module 1 (Standard 16 PD)^Inputs 16 PD^PI 4;
								.PD_5_IST_STROM  		:= TIID^Device 1 (EtherCAT)^=3400+FS2-16T1 (Bohraggr Schlüsselloch oben)^Module 1 (Standard 16 PD)^Inputs 16 PD^PI 5'}		
		e_Bohraggr_Schluessel_ob	AT%I*	: DUT_SEW_FU_PD_IN; 	// Schnittstelle zwischen SPS und FU
	 {attribute 'TcLinkTo' := '	.PD_1_Steuerwort  		:= TIID^Device 1 (EtherCAT)^=3400+FS2-16T1 (Bohraggr Schlüsselloch oben)^Module 1 (Standard 16 PD)^Outputs 16 PD^PO 1;
								.PD_2_Solldrehzahl  	:= TIID^Device 1 (EtherCAT)^=3400+FS2-16T1 (Bohraggr Schlüsselloch oben)^Module 1 (Standard 16 PD)^Outputs 16 PD^PO 2;
								.PD_3_Sollbeschleunigung:= TIID^Device 1 (EtherCAT)^=3400+FS2-16T1 (Bohraggr Schlüsselloch oben)^Module 1 (Standard 16 PD)^Outputs 16 PD^PO 3;
								.PD_4_Sollverzoegerung  := TIID^Device 1 (EtherCAT)^=3400+FS2-16T1 (Bohraggr Schlüsselloch oben)^Module 1 (Standard 16 PD)^Outputs 16 PD^PO 4;
								.PD_5_Digitalausgaenge  := TIID^Device 1 (EtherCAT)^=3400+FS2-16T1 (Bohraggr Schlüsselloch oben)^Module 1 (Standard 16 PD)^Outputs 16 PD^PO 5'}
		a_Bohraggr_Schluessel_ob	AT%Q*	: DUT_SEW_FU_PD_OUT;	// Schnittstelle zwischen SPS und FU


    // Eingaenge
    //_______________________________________________________

    // +FS1-3K5

        {attribute 'TcLinkTo' := 'TIID^Device 1 (EtherCAT)^+FS1-3K1 (BK1120)^+FS1-3K5 (EL1809)^Channel 12^Input'}
        e_FR_3400_Bohraggregat_7_Schluesselloch_oben_Stillstandserkennung_Motor_steht AT %I* : BOOL; (* =FR.3400 Bohraggregat 7 (Schlüsselloch oben) Stillstandserkennung Motor steht *)

    // +K110-1K2

        {attribute 'TcLinkTo' := 'TIID^Device 1 (EtherCAT)^+K110-1K1 (BK1120)^+K110-1K2 (EL1809)^Channel 14^Input'}
        e_FR_3400_Druecker_Schluesselloch_oben_Bohraggregat_7_Bohrhub_ist_oben AT %I* : BOOL; (* =FR.3400 Drücker/Schlüsselloch oben Bohraggregat 7 Bohrhub ist oben *)

        {attribute 'TcLinkTo' := 'TIID^Device 1 (EtherCAT)^+K110-1K1 (BK1120)^+K110-1K2 (EL1809)^Channel 15^Input'}
        e_FR_3400_Druecker_Schluesselloch_oben_Bohraggregat_7_Bohrhub_ist_unten AT %I* : BOOL; (* =FR.3400 Drücker/Schlüsselloch oben Bohraggregat 7 Bohrhub ist unten *)


    // Ausgaenge
    //_______________________________________________________

    // +K110-2K1

        {attribute 'TcLinkTo' := 'TIID^Device 1 (EtherCAT)^+K110-1K1 (BK1120)^+K110-2K1 (EL2809)^Channel 15^Output'}
        a_FR_3400_Druecker_Schluesselloch_oben_Bohraggregat_7_Bohrhub_heben AT %Q* : BOOL; (* =FR.3400 Drücker/Schlüsselloch oben Bohraggregat 7 Bohrhub heben *)

        {attribute 'TcLinkTo' := 'TIID^Device 1 (EtherCAT)^+K110-1K1 (BK1120)^+K110-2K1 (EL2809)^Channel 16^Output'}
        a_FR_3400_Druecker_Schluesselloch_oben_Bohraggregat_7_Bohrhub_senken AT %Q* : BOOL; (* =FR.3400 Drücker/Schlüsselloch oben Bohraggregat 7 Bohrhub senken *)
END_VAR

// ---- 3400_Bohraggregat/GVL_3400.TcGVL

VAR_GLOBAL
    // Achsen ***************************************************	
	X_Achse_steuern						: DUT_Achse_Steuern;	
	X_Achse_status						: DUT_Achse_Status;	
		                            	
	Y_Achse_steuern						: DUT_Achse_Steuern;		
	Y_Achse_status						: DUT_Achse_Status;		

    // Frequenzumrichter ****************************************
	Bohraggr_Schluessel_ob_steuern		: DUT_SEW_FU_Steuern;	
	Bohraggr_Schluessel_ob_status		: DUT_SEW_FU_Status;

    // Ventile **************************************************
    Schluessel_ob_Bohrhub          		: DUT_Ventil_sps;

    // interne Variablen ****************************************
    sk_Freigabe                         : BOOL;
    sk                                  : INT;
    transport_einfoerdern_bereit        : BOOL;
    transport_ausfoerdern_bereit        : BOOL;

    Tuer_Anwahl                         : BOOL;   // Signal Tür Anwahl, Tür soll geöffnet werden
    Tuer_Freigabe                       : BOOL;   // Signal Tür Freigabe, Tür kann geöffnet werden
END_VAR

// ---- 3510_Transport/GVL_3510.TcGVL

VAR_GLOBAL
    // Achsen ***************************************************
    //Achse_steuern                     : DUT_Achse_Steuern;
    //Achse_status                      : DUT_Achse_Status;

    // Frequenzumrichter ****************************************
	Trans_Schlossseite_steuern			: DUT_SEW_FU_Steuern;	
	Trans_Schlossseite_status			: DUT_SEW_FU_Status;
	
    // Ventile **************************************************
    Laengsanschl          				: DUT_Ventil_sps;
    Schienenklemm          				: DUT_Ventil_sps;

    // interne Variablen ****************************************
    sk_Freigabe                         : BOOL;
    sk                                  : INT;
    transport_einfoerdern_bereit        : BOOL;
    transport_ausfoerdern_bereit        : BOOL;

    Tuer_Anwahl                         : BOOL;   // Signal Tür Anwahl, Tür soll geöffnet werden
    Tuer_Freigabe                       : BOOL;   // Signal Tür Freigabe, Tür kann geöffnet werden
END_VAR

// ---- 3520_Transport/GVL_3520.TcGVL

VAR_GLOBAL
    // Achsen ***************************************************	
	Y_Achse_steuern						: DUT_Achse_Steuern;		
	Y_Achse_status						: DUT_Achse_Status;		

    // Frequenzumrichter ****************************************
	Trans_Bandseite_steuern				: DUT_SEW_FU_Steuern;	
	Trans_Bandseite_status				: DUT_SEW_FU_Status;

    // Ventile **************************************************
    Laengsanschl          				: DUT_Ventil_sps;
    Schienenklemm          				: DUT_Ventil_sps;

    // interne Variablen ****************************************
    sk_Freigabe                         : BOOL;
    sk                                  : INT;
    transport_einfoerdern_bereit        : BOOL;
    transport_ausfoerdern_bereit        : BOOL;

    Tuer_Anwahl                         : BOOL;   // Signal Tür Anwahl, Tür soll geöffnet werden
    Tuer_Freigabe                       : BOOL;   // Signal Tür Freigabe, Tür kann geöffnet werden
END_VAR

// ---- 3520_Transport/GVL_Visu_3520.TcGVL

VAR_GLOBAL
    KommAnVisu                 : INT;      (* Kommunikation an die Visualisierung *)
    KommVonVisu                : INT;      (* Kommunikation von der Visualisierung *)
    belegt                     : BOOL;     (* true = erzeugt Dummyteil, false = keine Auswirkungen (nur Handauflage) *)
    daten_gebucht              : BOOL;
    SteuerStatus               : DUT_Visu_SteuerStatus;

    // Frequenzumrichter
	Trans_Bandseite				: DUT_SEW_FU_Visu; 		//#Tab: 3520 Transport #Name: Transport Bandseite X-Achse

    // Servoregler
	Y_Achse						: DUT_Achse_Service;	//#Tab: 3520 Transport #Name: Y-Achse 

    // Ventile
	 Laengsanschl        		: DUT_Ventil_VISU;      //#Tab: 3520 Transport #Name: Bandseite Längsanschlag
	 Schienenklemm        		: DUT_Ventil_VISU;      //#Tab: 3520 Transport #Name: Schienenklemmung

END_VAR

VAR_GLOBAL PERSISTENT
    Schrittnummer              : INT;
    //Kopfdaten                : DUT_Kopfdaten;
    //Kopfdaten_default        : DUT_Kopfdaten;
    //Jobdaten                 : DUT_Jobdaten;
    //Jobdaten_default         : DUT_Jobdaten;

    //para_Vorlage             : REAL := 0.0; //#Typ: VParam #Tab:  #Name:  #Einheit:mm #Min: 1 #Max: 100 #Format:F1
END_VAR

// ---- 3530_Niederhalter/GVL_3530.TcGVL

VAR_GLOBAL
    // Achsen ***************************************************
    //Achse_steuern                     : DUT_Achse_Steuern;
    //Achse_status                      : DUT_Achse_Status;

    // Frequenzumrichter ****************************************
    //transport_steuern                 : DUT_SEW_FU_Steuern;
    //transport_status                  : DUT_SEW_FU_Status;

    // Ventile **************************************************
    Niederhalter          				: DUT_Ventil_sps;

    // interne Variablen ****************************************
    sk_Freigabe                         : BOOL;
    sk                                  : INT;
    transport_einfoerdern_bereit        : BOOL;
    transport_ausfoerdern_bereit        : BOOL;

    Tuer_Anwahl                         : BOOL;   // Signal Tür Anwahl, Tür soll geöffnet werden
    Tuer_Freigabe                       : BOOL;   // Signal Tür Freigabe, Tür kann geöffnet werden
END_VAR

// ---- 3540_Niederhalter/EAs_3540.TcGVL
{attribute 'qualified_only'}
{attribute 'linkalways'} 
VAR_GLOBAL

	// Servoregler *************************************************************************************************************************************************

	{attribute 'TcNcAxis':='=3540+FS2-11M1 (Y-Achse)'}	
	ea_Y_Achse					: Axis_ref;				// Schnittstellen Struktur zwischen NC<->SPS


    // Eingaenge
    //_______________________________________________________

    // +K110-1K3

        {attribute 'TcLinkTo' := 'TIID^Device 1 (EtherCAT)^+K110-1K1 (BK1120)^+K110-1K3 (EL1809)^Channel 6^Input'}
        e_FR_3540_Niederhalter_Bandseite_Niederhalter_Einlauf_ist_oben AT %I* : BOOL; (* =FR.3540 Niederhalter Bandseite Niederhalter Einlauf ist oben *)

        {attribute 'TcLinkTo' := 'TIID^Device 1 (EtherCAT)^+K110-1K1 (BK1120)^+K110-1K3 (EL1809)^Channel 7^Input'}
        e_FR_3540_Niederhalter_Bandseite_Niederhalter_Einlauf_ist_unten AT %I* : BOOL; (* =FR.3540 Niederhalter Bandseite Niederhalter Einlauf ist unten *)

        {attribute 'TcLinkTo' := 'TIID^Device 1 (EtherCAT)^+K110-1K1 (BK1120)^+K110-1K3 (EL1809)^Channel 8^Input'}
        e_FR_3540_Niederhalter_Bandseite_Niederhalter_Auslauf_ist_oben AT %I* : BOOL; (* =FR.3540 Niederhalter Bandseite Niederhalter Auslauf ist oben *)

        {attribute 'TcLinkTo' := 'TIID^Device 1 (EtherCAT)^+K110-1K1 (BK1120)^+K110-1K3 (EL1809)^Channel 9^Input'}
        e_FR_3540_Niederhalter_Bandseite_Niederhalter_Auslauf_ist_unten AT %I* : BOOL; (* =FR.3540 Niederhalter Bandseite Niederhalter Auslauf ist unten *)


    // Ausgaenge
    //_______________________________________________________

    // +K110-2K2

        {attribute 'TcLinkTo' := 'TIID^Device 1 (EtherCAT)^+K110-1K1 (BK1120)^+K110-2K2 (EL2809)^Channel 7^Output'}
        a_FR_3540_Niederhalter_Bandseite_Niederhalter_heben AT %Q* : BOOL; (* =FR.3540 Niederhalter Bandseite Niederhalter heben *)

        {attribute 'TcLinkTo' := 'TIID^Device 1 (EtherCAT)^+K110-1K1 (BK1120)^+K110-2K2 (EL2809)^Channel 8^Output'}
        a_FR_3540_Niederhalter_Bandseite_Niederhalter_senken AT %Q* : BOOL; (* =FR.3540 Niederhalter Bandseite Niederhalter senken *)
END_VAR

// ---- 0000/Ablauf_0000.TcPOU

PROGRAM Ablauf_0000
VAR
    // TODO: lokale Variablen fuer den Ablauf deklarieren
END_VAR


// TODO: Hauptprogramm-Code fuer Ablauf hier einfuegen


METHOD M_VisuKomm : BOOL
VAR_INPUT
    Nr          : INT;
END_VAR
VAR_IN_OUT
    anVisu      : INT;
    vonVisu     : INT;
END_VAR

VAR_INST
    result                  : INT;
    ton_DatenUngueltig      : TON;
    ton_DatenTimeout        : TON;
    sc                      : INT;
END_VAR

// Schnistelle zur VISU Kommunikation
// Starttrigger belegen als Antwort wird auf die 5= gut oder 9=schlecht gewartet.
// Kommunikationstimeout nach 5 Sekunden und wird automatisch wieder neugestartet

ton_DatenTimeout(IN:= anVisu <> 0 AND vonVisu = 0, PT:=T#3S);
ton_DatenUngueltig(IN:= sc = 20, PT:=T#500MS);

CASE sc OF
    0:  // Anfrage starten und auf Antwort warten
        anVisu := Nr;
        result := 0;
        IF vonVisu <> 0 THEN
            IF (vonVisu MOD Nr) = 5 THEN
                sc := 10;
            ELSIF (vonVisu MOD Nr) = 9 THEN
                sc := 20;
            END_IF
        ELSIF ton_DatenTimeout.Q THEN
            sc := 20;
        END_IF

    10: // Antwort 5 erhalten
        anVisu := 0;
        IF vonVisu = 0 THEN
            M_VisuKomm := TRUE;
            result := 1;
            sc := 0;
        END_IF

    20: // Timeout, 1 Sekunde warten und erneut antriggern
        IF ton_DatenUngueltig.Q THEN
            anVisu := 0;
            IF vonVisu = 0 THEN
                result := -1;
                sc := 0;
            END_IF
        END_IF

END_CASE
END_METHOD


METHOD M_VisuKommInt : INT
VAR_INPUT
    Nr          : INT;
END_VAR
VAR_IN_OUT
    anVisu      : INT;
    vonVisu     : INT;
END_VAR

VAR_INST
    result                  : INT;
    ton_DatenUngueltig      : TON;
    ton_DatenTimeout        : TON;
    sc                      : INT;
END_VAR

// Schnistelle zur VISU Kommunikation
// Starttrigger belegen als Antwort wird auf die 5= gut oder 9=schlecht gewartet.
// Kommunikationstimeout nach 5 Sekunden und wird automatisch wieder neugestartet

ton_DatenTimeout(IN:= anVisu <> 0 AND vonVisu = 0, PT:=T#3S);
ton_DatenUngueltig(IN:= anVisu = 0 AND vonVisu = 0, PT:=T#500MS);

CASE sc OF
    0:  // Anfrage starten und auf Antwort warten
        anVisu := Nr;
        result := 0;
        IF vonVisu <> 0 THEN
            IF (vonVisu MOD Nr) = 5 THEN
                sc := 10;
            ELSIF (vonVisu MOD Nr) = 9 THEN
                sc := 15;
            END_IF
        ELSIF ton_DatenTimeout.Q THEN
            sc := 20;
        END_IF

    10: // Antwort 5 erhalten (OK)
        anVisu := 0;
        IF vonVisu = 0 THEN
            M_VisuKommInt := 1;
            result := 1;
            sc := 0;
        END_IF

    15: // Antwort 9 erhalten (Fehler)
        anVisu := 0;
        IF vonVisu = 0 THEN
            M_VisuKommInt := -1;
            result := 1;
            sc := 0;
        END_IF

    20: // Timeout, 1 Sekunde warten und erneut antriggern
        anVisu := 0;
        IF vonVisu = 0 THEN
            result := -1;
            IF ton_DatenUngueltig.Q THEN
                sc := 0;
            END_IF
        END_IF

END_CASE
END_METHOD

END_PROGRAM

// ---- 3100_Bohraggregat/Ablauf_3100.TcPOU

PROGRAM Ablauf_3100
VAR
    // TODO: lokale Variablen fuer den Ablauf deklarieren
END_VAR


// TODO: Hauptprogramm-Code fuer Ablauf hier einfuegen


METHOD M_VisuKomm : BOOL
VAR_INPUT
    Nr          : INT;
END_VAR
VAR_IN_OUT
    anVisu      : INT;
    vonVisu     : INT;
END_VAR

VAR_INST
    result                  : INT;
    ton_DatenUngueltig      : TON;
    ton_DatenTimeout        : TON;
    sc                      : INT;
END_VAR

// Schnistelle zur VISU Kommunikation
// Starttrigger belegen als Antwort wird auf die 5= gut oder 9=schlecht gewartet.
// Kommunikationstimeout nach 5 Sekunden und wird automatisch wieder neugestartet

ton_DatenTimeout(IN:= anVisu <> 0 AND vonVisu = 0, PT:=T#3S);
ton_DatenUngueltig(IN:= sc = 20, PT:=T#500MS);

CASE sc OF
    0:  // Anfrage starten und auf Antwort warten
        anVisu := Nr;
        result := 0;
        IF vonVisu <> 0 THEN
            IF (vonVisu MOD Nr) = 5 THEN
                sc := 10;
            ELSIF (vonVisu MOD Nr) = 9 THEN
                sc := 20;
            END_IF
        ELSIF ton_DatenTimeout.Q THEN
            sc := 20;
        END_IF

    10: // Antwort 5 erhalten
        anVisu := 0;
        IF vonVisu = 0 THEN
            M_VisuKomm := TRUE;
            result := 1;
            sc := 0;
        END_IF

    20: // Timeout, 1 Sekunde warten und erneut antriggern
        IF ton_DatenUngueltig.Q THEN
            anVisu := 0;
            IF vonVisu = 0 THEN
                result := -1;
                sc := 0;
            END_IF
        END_IF

END_CASE
END_METHOD


METHOD M_VisuKommInt : INT
VAR_INPUT
    Nr          : INT;
END_VAR
VAR_IN_OUT
    anVisu      : INT;
    vonVisu     : INT;
END_VAR

VAR_INST
    result                  : INT;
    ton_DatenUngueltig      : TON;
    ton_DatenTimeout        : TON;
    sc                      : INT;
END_VAR

// Schnistelle zur VISU Kommunikation
// Starttrigger belegen als Antwort wird auf die 5= gut oder 9=schlecht gewartet.
// Kommunikationstimeout nach 5 Sekunden und wird automatisch wieder neugestartet

ton_DatenTimeout(IN:= anVisu <> 0 AND vonVisu = 0, PT:=T#3S);
ton_DatenUngueltig(IN:= anVisu = 0 AND vonVisu = 0, PT:=T#500MS);

CASE sc OF
    0:  // Anfrage starten und auf Antwort warten
        anVisu := Nr;
        result := 0;
        IF vonVisu <> 0 THEN
            IF (vonVisu MOD Nr) = 5 THEN
                sc := 10;
            ELSIF (vonVisu MOD Nr) = 9 THEN
                sc := 15;
            END_IF
        ELSIF ton_DatenTimeout.Q THEN
            sc := 20;
        END_IF

    10: // Antwort 5 erhalten (OK)
        anVisu := 0;
        IF vonVisu = 0 THEN
            M_VisuKommInt := 1;
            result := 1;
            sc := 0;
        END_IF

    15: // Antwort 9 erhalten (Fehler)
        anVisu := 0;
        IF vonVisu = 0 THEN
            M_VisuKommInt := -1;
            result := 1;
            sc := 0;
        END_IF

    20: // Timeout, 1 Sekunde warten und erneut antriggern
        anVisu := 0;
        IF vonVisu = 0 THEN
            result := -1;
            IF ton_DatenUngueltig.Q THEN
                sc := 0;
            END_IF
        END_IF

END_CASE
END_METHOD

END_PROGRAM

// ---- 3300_Bohraggregat/Ablauf_3300.TcPOU

PROGRAM Ablauf_3300
VAR
    // TODO: lokale Variablen fuer den Ablauf deklarieren
END_VAR


// TODO: Hauptprogramm-Code fuer Ablauf hier einfuegen


METHOD M_VisuKomm : BOOL
VAR_INPUT
    Nr          : INT;
END_VAR
VAR_IN_OUT
    anVisu      : INT;
    vonVisu     : INT;
END_VAR

VAR_INST
    result                  : INT;
    ton_DatenUngueltig      : TON;
    ton_DatenTimeout        : TON;
    sc                      : INT;
END_VAR

// Schnistelle zur VISU Kommunikation
// Starttrigger belegen als Antwort wird auf die 5= gut oder 9=schlecht gewartet.
// Kommunikationstimeout nach 5 Sekunden und wird automatisch wieder neugestartet

ton_DatenTimeout(IN:= anVisu <> 0 AND vonVisu = 0, PT:=T#3S);
ton_DatenUngueltig(IN:= sc = 20, PT:=T#500MS);

CASE sc OF
    0:  // Anfrage starten und auf Antwort warten
        anVisu := Nr;
        result := 0;
        IF vonVisu <> 0 THEN
            IF (vonVisu MOD Nr) = 5 THEN
                sc := 10;
            ELSIF (vonVisu MOD Nr) = 9 THEN
                sc := 20;
            END_IF
        ELSIF ton_DatenTimeout.Q THEN
            sc := 20;
        END_IF

    10: // Antwort 5 erhalten
        anVisu := 0;
        IF vonVisu = 0 THEN
            M_VisuKomm := TRUE;
            result := 1;
            sc := 0;
        END_IF

    20: // Timeout, 1 Sekunde warten und erneut antriggern
        IF ton_DatenUngueltig.Q THEN
            anVisu := 0;
            IF vonVisu = 0 THEN
                result := -1;
                sc := 0;
            END_IF
        END_IF

END_CASE
END_METHOD


METHOD M_VisuKommInt : INT
VAR_INPUT
    Nr          : INT;
END_VAR
VAR_IN_OUT
    anVisu      : INT;
    vonVisu     : INT;
END_VAR

VAR_INST
    result                  : INT;
    ton_DatenUngueltig      : TON;
    ton_DatenTimeout        : TON;
    sc                      : INT;
END_VAR

// Schnistelle zur VISU Kommunikation
// Starttrigger belegen als Antwort wird auf die 5= gut oder 9=schlecht gewartet.
// Kommunikationstimeout nach 5 Sekunden und wird automatisch wieder neugestartet

ton_DatenTimeout(IN:= anVisu <> 0 AND vonVisu = 0, PT:=T#3S);
ton_DatenUngueltig(IN:= anVisu = 0 AND vonVisu = 0, PT:=T#500MS);

CASE sc OF
    0:  // Anfrage starten und auf Antwort warten
        anVisu := Nr;
        result := 0;
        IF vonVisu <> 0 THEN
            IF (vonVisu MOD Nr) = 5 THEN
                sc := 10;
            ELSIF (vonVisu MOD Nr) = 9 THEN
                sc := 15;
            END_IF
        ELSIF ton_DatenTimeout.Q THEN
            sc := 20;
        END_IF

    10: // Antwort 5 erhalten (OK)
        anVisu := 0;
        IF vonVisu = 0 THEN
            M_VisuKommInt := 1;
            result := 1;
            sc := 0;
        END_IF

    15: // Antwort 9 erhalten (Fehler)
        anVisu := 0;
        IF vonVisu = 0 THEN
            M_VisuKommInt := -1;
            result := 1;
            sc := 0;
        END_IF

    20: // Timeout, 1 Sekunde warten und erneut antriggern
        anVisu := 0;
        IF vonVisu = 0 THEN
            result := -1;
            IF ton_DatenUngueltig.Q THEN
                sc := 0;
            END_IF
        END_IF

END_CASE
END_METHOD

END_PROGRAM

// ---- 3300_Bohraggregat/Hardware_3300.TcPOU

PROGRAM Hardware_3300
VAR
    // Servos *********************************************************************
	fbX_Achse										: FB_Achse_NC_PTP_Beckhoff; 
	fbY_Achse										: FB_Achse_NC_PTP_Beckhoff; 

    // Frequenzumrichter **********************************************************
	fbBohraggr_Schluessel_un						: FB_SEW_MOVITRAC_C_CoE;

    // Sensorik *******************************************************************
    fbStillBohraggr_Schluessel_un          			: FB_Belegt;

    // Ventile ********************************************************************
    fbSchluessel_un_Bohrhub                			: FB_Ventil_V2;

    // ***** Hilfsmerker***********************************************************
    (*
        Ventile sind über den DUT_Ventil_para vorparametriert
                ueberwachung_vor_aktiv    : BOOL := TRUE;   // 0 = Endlagenüberwachung vor deaktiviert
                ueberwachung_zur_aktiv    : BOOL := TRUE;   // 0 = Endlagenüberwachung zurück deaktiviert
                ausgang_vor_halten        : BOOL := FALSE;  // 1 = Ausgang immer Ein, sonst 0 in Endlage/1 nicht in Endlage
                ausgang_zur_halten        : BOOL := FALSE;  // 1 = Ausgang immer Ein, sonst 0 in Endlage/1 nicht in Endlage
                entprellen_vor_aktiv      : BOOL := TRUE;   // 0 = Endlage sofort überwachen wenn einmal erreicht
                entprellen_zur_aktiv      : BOOL := TRUE;   // 0 = Endlage sofort überwachen wenn einmal erreicht
                ueberwachungszeit_vor     : TIME := T#10S;  // Überwachungszeit in ms (0-30000ms)
                ueberwachungszeit_zur     : TIME := T#10S;  // Überwachungszeit in ms (0-30000ms)
                entprellungszeit_vor      : TIME := T#50MS; // Entprellungszeit in ms (0-10000ms)
                entprellungszeit_zur      : TIME := T#50MS; // Entprellungszeit in ms (0-10000ms)

        falls etwas anderes gewünscht ist, kann man gezielt für das Ventil die Parameter anpassen
        Beispiel:   ***.para.ausgang_vor_halten := TRUE;
                    ***.para.entprellungszeit_vor := T#100MS;
    *)
END_VAR


// Aktionen aufrufen
//_________________________________________________
	A_Sensorik();
	A_Umrichter();
	A_Ventile();
	A_Servo();

ACTION A_Sensorik:
					
// ***** Sensorik entprellen *********************************************************
	//********************************************************************************
fbStillBohraggr_Schluessel_un	(	in_Sensor:=,
									in_zeit_aus:=T#100MS,
									in_zeit_aus:=T#100MS,
									Q=>);
END_ACTION

ACTION A_Servo:
					
// ***** Servoregler *****************************************************************
	//********************************************************************************
	GVL_3300.X_Achse_steuern.Reglersperre	:= FALSE;
	GVL_3300.X_Achse_steuern.Freigabe 		:= FALSE;
	
	fbX_Achse(
	in_Reglersperre				:= GVL_3300.X_Achse_steuern.Reglersperre, 
	in_Freigabe					:= GVL_3300.X_Achse_steuern.Freigabe,
	in_Reset					:= GVL_Visu_3300.SteuerStatus.reset   
								OR GVL_0000.stoerung_quitt,                      
	in_Hand						:= GVL_Visu_3300.SteuerStatus.hand,              
	in_Auto						:= GVL_Visu_3300.SteuerStatus.auto,                 
	in_Auto_Override			:= GVL_Visu_0000.override,    
	in_Auto_pos					:= , 
	in_PosFenster				:= 0.05, 
	in_Ref_pos					:= 0.0, 
	in_HomingOption				:= , 
	in_EndlageRef				:= , 
	in_DirRef					:= , 
	in_PosEa					:= ,                                       
	out_ist_pos					=> GVL_3300.X_Achse_status.ist_pos, 
	out_in_pos					=> GVL_3300.X_Achse_status.in_pos,   
	out_ziel_pos				=> GVL_3300.X_Achse_status.ziel_pos, 
	out_nicht_ref				=> GVL_3300.X_Achse_status.nicht_ref,      
	out_bremse					=> GVL_3300.X_Achse_status.bremse,           
	out_Achs_Status				=> GVL_3300.X_Achse_status.Achs_Status,  
	inout_NC					:= EAs_3300.ea_X_Achse, 
	inout_service				:= GVL_Visu_3300.X_Achse, 
	inout_Ref_start				:= GVL_3300.X_Achse_steuern.Ref_start, 
	inout_Auto_start			:= GVL_3300.X_Achse_steuern.Auto_start, 
	inout_Auto_stop				:= GVL_3300.X_Achse_steuern.Auto_stop);
	
	GVL_Meldungen.Diagnose_3000.Nr_028	:= fbX_Achse.out_Achs_ErrorID;	
	GVL_Meldungen.Meldungen_3000.Nr_028 := fbX_Achse.out_Achs_Error OR fbX_Achse.out_FB_Error OR fbX_Achse.out_Achs_ErrorID <> 0;		
	GVL_Meldungen.Meldungen_3000.Nr_029 := FALSE;
	GVL_Meldungen.Meldungen_3000.Nr_030 := FALSE;
	//********************************************************************************
					
					
	GVL_3300.Y_Achse_steuern.Reglersperre	:= FALSE;
	GVL_3300.Y_Achse_steuern.Freigabe 		:= FALSE;
	
	fbY_Achse(
	in_Reglersperre				:= GVL_3300.Y_Achse_steuern.Reglersperre, 
	in_Freigabe					:= GVL_3300.Y_Achse_steuern.Freigabe,
	in_Reset					:= GVL_Visu_3300.SteuerStatus.reset   
								OR GVL_0000.stoerung_quitt,                      
	in_Hand						:= GVL_Visu_3300.SteuerStatus.hand,              
	in_Auto						:= GVL_Visu_3300.SteuerStatus.auto,                 
	in_Auto_Override			:= GVL_Visu_0000.override,    
	in_Auto_pos					:= , 
	in_PosFenster				:= 0.05, 
	in_Ref_pos					:= 0.0, 
	in_HomingOption				:= , 
	in_EndlageRef				:= , 
	in_DirRef					:= , 
	in_PosEa					:= ,                                       
	out_ist_pos					=> GVL_3300.Y_Achse_status.ist_pos, 
	out_in_pos					=> GVL_3300.Y_Achse_status.in_pos,   
	out_ziel_pos				=> GVL_3300.Y_Achse_status.ziel_pos, 
	out_nicht_ref				=> GVL_3300.Y_Achse_status.nicht_ref,      
	out_bremse					=> GVL_3300.Y_Achse_status.bremse,           
	out_Achs_Status				=> GVL_3300.Y_Achse_status.Achs_Status,  
	inout_NC					:= EAs_3300.ea_Y_Achse, 
	inout_service				:= GVL_Visu_3300.Y_Achse, 
	inout_Ref_start				:= GVL_3300.Y_Achse_steuern.Ref_start, 
	inout_Auto_start			:= GVL_3300.Y_Achse_steuern.Auto_start, 
	inout_Auto_stop				:= GVL_3300.Y_Achse_steuern.Auto_stop);
	
	GVL_Meldungen.Diagnose_3000.Nr_031	:= fbY_Achse.out_Achs_ErrorID;	
	GVL_Meldungen.Meldungen_3000.Nr_031 := fbY_Achse.out_Achs_Error OR fbY_Achse.out_FB_Error OR fbY_Achse.out_Achs_ErrorID <> 0;		
	GVL_Meldungen.Meldungen_3000.Nr_032 := FALSE;
	GVL_Meldungen.Meldungen_3000.Nr_033 := FALSE;
END_ACTION

ACTION A_Umrichter:
	
// ***** Frequenzumrichter ******************************************************
// ******************************************************************************
				
	GVL_Visu_3300.Bohraggr_Schluessel_un	.Para.Speed_Hand		:= 0;
	GVL_Visu_3300.Bohraggr_Schluessel_un	.Para.Beschleunigung 	:= 0;
	GVL_Visu_3300.Bohraggr_Schluessel_un	.Para.Verzoegerung 		:= 0;
	GVL_Visu_3300.Bohraggr_Schluessel_un	.Para.Einheit			:= 1;

	fbBohraggr_Schluessel_un	(	PD_IN	:=EAs_3300.e_Bohraggr_Schluessel_un	,
			IN_ReglerSperre			:=,
			IN_SteuerStatus			:=GVL_Visu_3300.SteuerStatus,
			IN_Ethercat_Adresse		:=,
			IN_Ethercat_Name		:='',
			IN_QUITTIEREN			:= GVL_0000.stoerung_quitt,
			IN_OVERRIDE				:= GVL_Visu_0000.override,
			PD_OUT					=> EAs_3300.a_Bohraggr_Schluessel_un	,
			OUT_Stoerung			=> GVL_Meldungen.Meldungen_3000.Nr_006,
			OUT_Fehlernummer		=> GVL_Meldungen.Diagnose_3000.Nr_006,
			OUT_Status				=> GVL_3300.Bohraggr_Schluessel_un_status,
			inout_visu				:= GVL_Visu_3300.Bohraggr_Schluessel_un	,
			inout_steuern			:= GVL_3300.Bohraggr_Schluessel_un_steuern);
	
			GVL_3300.Bohraggr_Schluessel_un_steuern.vor := FALSE;
			GVL_3300.Bohraggr_Schluessel_un_steuern.zur := FALSE;
			GVL_3300.Bohraggr_Schluessel_un_steuern.speed := 0;
END_ACTION

ACTION A_Ventile:
	
// ***** Ventile *********************************************************************
	//********************************************************************************	
	
	GVL_Visu_3300.Schluessel_un_Bohrhub.para.ausgang_vor_halten:=TRUE;	
	GVL_Visu_3300.Schluessel_un_Bohrhub.para.ausgang_zur_halten:=TRUE;	
	GVL_Visu_3300.Schluessel_un_Bohrhub.para.ueberwachung_vor_aktiv:=TRUE;	
	GVL_Visu_3300.Schluessel_un_Bohrhub.para.ueberwachung_zur_aktiv:=TRUE;	
	GVL_Visu_3300.Schluessel_un_Bohrhub.para.entprellungszeit_vor:=T#50S;	
	GVL_Visu_3300.Schluessel_un_Bohrhub.para.entprellungszeit_zur:=T#50MS;	
	fbSchluessel_un_Bohrhub (	in_endlage_vor:= EAs_3300.e_FR_3300_Druecker_Schluesselloch_unten_Bohraggregat_6_Bohrhub_ist_oben,
								in_endlage_zur:= EAs_3300.e_FR_3300_Druecker_Schluesselloch_unten_Bohraggregat_6_Bohrhub_ist_unten,
								in_hand:=GVL_Visu_3300.SteuerStatus.hand,
								in_auto:=GVL_Visu_3300.SteuerStatus.auto,
								in_quit:=GVL_Visu_3300.SteuerStatus.reset 
								OR GVL_0000.stoerung_quitt,
								out_vor=>EAs_3300.a_FR_3300_Druecker_Schluesselloch_unten_Bohraggregat_6_Bohrhub_heben,
								out_zur=>EAs_3300.a_FR_3300_Druecker_Schluesselloch_unten_Bohraggregat_6_Bohrhub_senken,
								out_stoerung_vor=> GVL_Meldungen.Meldungen_3000.Nr_067,
								out_stoerung_zur=> GVL_Meldungen.Meldungen_3000.Nr_068,
								out_stoerung_vorzur=> GVL_Meldungen.Meldungen_3000.Nr_069,
								inout_ansteuerung:=GVL_3300.Schluessel_un_Bohrhub ,
								inout_visu:=GVL_Visu_3300.Schluessel_un_Bohrhub );
END_ACTION

END_PROGRAM

// ---- SRT_Allgemein/0010_Bausteine_mitDuts/POUs/FU_SEW/Movi_C/FB_SEW_MOVITRAC_C_COE.TcPOU
FUNCTION_BLOCK FB_SEW_MOVITRAC_C_COE
VAR_INPUT
	PD_IN					:DUT_SEW_FU_PD_IN;
	IN_REGLERSPERRE			:BOOL;	(* 1= Regler sperren *)
	IN_STEUERSTATUS			:DUT_VISU_Steuerstatus;
	IN_ETHERCAT_ADRESSE		:UINT;
	IN_ETHERCAT_NAME		:STRING;
	IN_OVERRIDE				:INT;
	IN_QUITTIEREN			: BOOL;
END_VAR
VAR_OUTPUT
	PD_OUT					:DUT_SEW_FU_PD_OUT;
	OUT_STOERUNG			:BOOL;	(* Umrichter meldet Störung *)
	OUT_FEHLERNUMMER		:DINT;	(* Fehlernummer *)
	OUT_STATUS				:DUT_SEW_FU_STATUS;
	//OUT_WARNUNG				:BOOL;
END_VAR
VAR_TEMP
	

END_VAR
VAR_IN_OUT
inout_Visu					:DUT_SEW_FU_Visu;
inout_steuern				:DUT_SEW_FU_Steuern;
END_VAR


VAR
	reglersperre			:BOOL;	(* BIT 0: Reglersperre 0 = Freigabe 1 = Regler sperren, Bremse aktivieren *)
	freigabe_stop			:BOOL;	(* BIT 1: Freigabe/Schnellstopp 0 = Schnellstopp 1 = Freigabe *)
	freigabe_halt			:BOOL;	(* BIT 2: Freigabe/Halt 0 = Halt an Integratorrampe oder Prozess-Rampe 1 = Freigabe *)
	reserve_3_1				:BOOL;	(* BIT 3: Reserviert (Reservierte Bits sind generell auf Null zu setzen!) *)
	reserve_4_1				:BOOL;	(* BIT 4: Reserviert (Reservierte Bits sind generell auf Null zu setzen!) *)
	reserve_5_1				:BOOL;	(* BIT 5: Reserviert (Reservierte Bits sind generell auf Null zu setzen!) *)
	reset					:BOOL;	(* Bit 6: Reset 0 = nicht aktiv 0 -> 1 = anstehende Störung zurücksetzen *)
	reserve_7_1				:BOOL;	(* BIT 7: Reserviert (Reservierte Bits sind generell auf Null zu setzen!) *)
	drehrichtung_motorpoti	:BOOL;	(* BIT 8: Drehrichtung für Motorpoti 0 = Drehrichtung RECHTS 1 = Drehrichtung LINKS *)
	motorpoti_auf			:BOOL;	(* BIT 9 und 10: Motorpoti Hochlauf,Motorpoti Tieflauf 0 0 = keine Änderung *)
	motorpoti_ab			:BOOL;	(*  1 0 = ab 0 1 = auf 1 1 = keine Änderung *)
	n11_n21					:BOOL;	(* BIT 11 und 12:Anwahl der internen Festsollwerte0 0 = Drehzahl-Sollwert über Prozess-Ausgangsdatenwort 2 *)
	n12_n22					:BOOL;	(* 0 1 = interner Sollwert n11 (n21) *)
	sollwert_umschaltung	:BOOL;	(* BIT 13: Festsollwert-Umschaltung 0 = Festsollwerte des aktivn Parameter über Bit 11/12 anwählbar 1 = Festsollwerte des anderen Parameter anwählbar *)
	reserve_14				:BOOL;	(* BIT 14: Reserviert (Reservierte Bits sind generell auf Null zu setzen!) *)
	reserve_15				:BOOL;	(* BIT 14: Reserviert (Reservierte Bits sind generell auf Null zu setzen!) *)


	DREHZAHL				:REAL;
	TEMP_IST_DREHZAHL_DINT	:DINT;
	TEMP_DREHZAHL			:REAL;
	TEMP_DREHZAHL_SOLL		:WORD;
	endstufe_freigegeben	:BOOL;	(* BIT 0: Endstufe freigegeben 0 = Endstufe ist gesperrt (hochohmig) 1 = Endstufe ist freigegeben *)
	umrichter_bb			:BOOL;	(* BIT 1: Umrichter betriebsbereit 0 = Umrichter nicht betriebsbereit (z. B. Fehler) 1 = Umrichter betriebsbereit *)
	pa_daten_freigeben		:BOOL;	(* BIT 2: PA-Daten freigegeben 0 = PA-Daten gesperrt 1 = PA-Daten freigegeben *)
	reserve_3				:BOOL;	(*  Reserve Bit ist immer auf null zusetzen *)
	reserve_4				:BOOL;	(*  Reserve Bit ist immer auf null zusetzen *)
	stoerung				:BOOL;	(*  BIT 5: Störung/Warnung 0 = keine Störung/Warnung 1 = Störung/Warnung liegt an *)
	reserver_6				:BOOL;	(*  Reserve Bit ist immer auf null zusetzen *)
	fehlernummer			:BYTE;	(*  Byte 2: Gerätezustand/ Fehlernummer *)
	steuerbyte_1			:BYTE;
	steuerbyte_2			:BYTE;
	STO_inaktiv				:BOOL;
	bremse_geoeffnet		: BOOL;
	motor_dreht				: BOOL;

	start_stop				:BOOL;
	jog_pos					:BOOL;
	jog_neg					:BOOL;
	hm_hand_vor: BOOL;
	hm_hand_zur: BOOL;
	
	//---COE
	CoE_ReadAndWrite		:FB_SEW_CoE;
	//Flankenmerker
	pFL_btnLesen			:R_TRIG;
	pFL_btnSchreiben		:R_TRIG;
	nFL_CoEBetriabsart		:F_TRIG;
	nFl_Hand				:F_TRIG;
	nFl_Auto				:F_TRIG;
	
	//Timer
	tofLesenErfolgreich			:TOF;
	tofLesenFehlgeschlagen		:TOF;
	tofSchreibenErfolgreich		:TOF;
	tofSchreibenFehlgeschlagen	:TOF;
	
	//BOOLS
	aktuellLesen				:BOOL;
	LesenErfolgreich			:BOOL;
	LesenFehlgeschlagen			:BOOL;
	aktuellSchreiben			:BOOL;
	SchreibenErfolgreich		:BOOL;
	SchreibenFehlgeschlagen		:BOOL;
	keinTimerAktiv				:BOOL;
	
	
END_VAR


//---Aufruf Statuswort auslesen
Read_Statuswort();

//--- Aufruf Kommunikation zur SPS
ComToSPS();

//--- Aufruf Rampen
Rampen();

//--- Aufruf Handbetrieb
IF in_Steuerstatus.hand
THEN
// COE
	CoE();
	Handbetrieb();
ELSIF	
//--- Aufruf Automatikbetrieb
	in_Steuerstatus.auto
THEN	
	Automatikbetrieb();
END_IF

// Aufruf Freigaben
Freigaben();

//Aufruf Fehlerhandling
Fehlerhandling();

// Aufruf Steuerwort schreiben
Write_Steuerwort();

// Beim Verlassen der Betriebsart werte zurücksetzen
Betriebsart_zuruecksetzen();

//Zyklisch Start etc zurücksetzen
//inout_steuern.vor 		:=FALSE;
//inout_steuern.zur 		:=FALSE;
//inout_visu.plus_start	:=FALSE;
//inout_visu.minus_stop	:=FALSE;

ACTION Automatikbetrieb:
//===========================================
//###	Automatikgeschwinidgkeit schreiben	###
//===========================================


//---Geschwinidgkeit berechnen

TEMP_DREHZAHL_SOLL:= REAL_TO_WORD(inout_steuern.speed / 10 * IN_OVERRIDE);

//---PD-Sollgeschwinidgkeit beschreiben---

	IF  (inout_steuern.vor AND NOT inout_Visu.Para.Drehtausch)
		OR  (inout_steuern.zur AND inout_Visu.Para.Drehtausch)
	THEN
		PD_OUT.PD_2_Solldrehzahl:= TEMP_DREHZAHL_SOLL; 
		
	ELSIF (inout_steuern.zur AND NOT inout_Visu.Para.Drehtausch)
		OR  (inout_steuern.vor AND inout_Visu.Para.Drehtausch)
	THEN	
		PD_OUT.PD_2_Solldrehzahl:= TEMP_DREHZAHL_SOLL*-1; 
	END_IF


// Startbit 	
start_stop :=  inout_steuern.vor
				OR inout_steuern.zur;
END_ACTION

ACTION Betriebsart_zuruecksetzen:
// Beim Verlassen der Betriebsart werte zurücksetzen


nFl_Hand(CLK:=in_Steuerstatus.hand);
nFl_Auto(CLK:=in_Steuerstatus.auto_aktiv);


IF nFl_Hand.Q
THEN
	PD_out.PD_2_Solldrehzahl:=0;
	inout_Visu.betriebsart	:=0;
	jog_pos 				:=FALSE;
	jog_neg 				:=FALSE;
	start_stop				:=FALSE;
END_IF

IF nFl_Auto.Q
THEN
	PD_out.PD_2_Solldrehzahl:=0;
	start_stop				:=FALSE;
END_IF
END_ACTION

ACTION CoE:
//-------------------------------------
//Bausteinaufruf CoE
//-------------------------------------	
CoE_ReadAndWrite(I_sBMK:=IN_ETHERCAT_NAME,
				I_nEcSlaveAddr:=IN_ETHERCAT_ADRESSE,
				I_bReset:= inout_Visu.betriebsart<>5);
				
Status_CoE();

//-------------------------------------
//Button zurücksetzen
//-------------------------------------	
pFL_btnLesen(CLK:=inout_Visu.plus_start);
pFL_btnSchreiben(CLK:=inout_visu.minus_stop);
nFL_CoEBetriabsart(CLK:=inout_Visu.betriebsart=5);

IF pFL_btnLesen.Q
THEN
	inout_Visu.minus_stop:=FALSE;
	CoE_ReadAndWrite.I_bStartWriteFromCSV:=FALSE;
END_IF

IF pFL_btnSchreiben.Q
THEN
	inout_Visu.plus_start:=FALSE;
	CoE_ReadAndWrite.I_bStartRead:=FALSE;
END_IF

IF nFL_CoEBetriabsart.Q
THEN
	inout_Visu.minus_stop:=FALSE;
	inout_Visu.plus_start:=FALSE;
	CoE_ReadAndWrite.I_bStartWriteFromCSV:=FALSE;
	CoE_ReadAndWrite.I_bStartRead:=FALSE;
END_IF

//-------------------------------------
//FU->CSV
//-------------------------------------	
// Start Lesen			
IF inout_Visu.betriebsart = 5
	AND pFL_btnLesen.Q
THEN
	CoE_ReadAndWrite.I_bStartRead:=TRUE;
END_IF



//-------------------------------------
//CSV->FU
//-------------------------------------
//Start Schreiben
IF inout_Visu.betriebsart = 5
	AND inout_Visu.minus_stop
THEN
	CoE_ReadAndWrite.I_bStartWriteFromCSV:=TRUE;
END_IF

//Button zurücksetzen
IF CoE_ReadAndWrite.Q_bBusy
	OR CoE_ReadAndWrite.Q_bError
THEN
	inout_Visu.plus_start:=FALSE;
	inout_Visu.minus_stop:=FALSE;
END_IF

//-------------------------------------
//Status zuweisen und Start zurücksetzen
//-------------------------------------
//Timer
tofLesenErfolgreich			(PT:=T#3S);
tofLesenFehlgeschlagen		(PT:=T#3S);
tofSchreibenErfolgreich		(PT:=T#3S);
tofSchreibenFehlgeschlagen	(PT:=T#3S);

//Aktuellen Status oder Timer Starten
IF aktuellLesen								//akteuell Lesen
THEN
	inout_Visu.diagnose:=300;
ELSIF
	aktuellSchreiben						//aktuell Schreiben
THEN
	inout_Visu.diagnose:=306;
ELSIF	
	LesenErfolgreich						//Lesen erfolgreich
THEN
	tofLesenErfolgreich.IN:=TRUE;
	CoE_ReadAndWrite.I_bStartRead:=FALSE;
ELSIF
	LesenFehlgeschlagen						//Lesen fehlgeschlagen
THEN
	tofLesenFehlgeschlagen.IN:=TRUE;

ELSIF
	SchreibenErfolgreich					//Schreiben erfolgreich
THEN
	tofSchreibenErfolgreich.IN :=TRUE;
	CoE_ReadAndWrite.I_bStartWriteFromCSV:=FALSE;
ELSIF
	SchreibenFehlgeschlagen					//Schreiben fehlgeschlagen
THEN
	tofSchreibenFehlgeschlagen.IN :=TRUE;
ELSIF
	keinTimerAktiv
	AND inout_Visu.betriebsart = 5
THEN
	inout_Visu.diagnose:=0;
END_IF

//Status von Timer und Timer zurücksetzen
IF tofLesenErfolgreich.Q				//TOF Lesen erfolgreich
THEN
	tofLesenErfolgreich.IN:=FALSE;
	inout_Visu.diagnose:=301;
END_IF

IF tofLesenFehlgeschlagen.Q				//TOF Lesen fehlgeschlagen
THEN
	CoE_ReadAndWrite.I_bStartRead:=FALSE;
	tofLesenFehlgeschlagen.IN:=FALSE;
	inout_Visu.diagnose:=302;
END_IF

IF tofSchreibenErfolgreich.Q			//TOF Schreiben erfolgreich
THEN
	tofSchreibenErfolgreich.IN:=FALSE;
	inout_Visu.diagnose:=307;
END_IF

IF tofSchreibenFehlgeschlagen.Q			//TOF Schreiben fehlgeschlagen
THEN
	CoE_ReadAndWrite.I_bStartWriteFromCSV:=FALSE;	
	tofSchreibenFehlgeschlagen.IN:=FALSE;
	inout_Visu.diagnose:=308;
END_IF

keinTimerAktiv:= NOT (	tofLesenErfolgreich.Q
					 OR tofLesenFehlgeschlagen.Q	
					 OR tofSchreibenErfolgreich.Q
					 OR tofSchreibenFehlgeschlagen.Q);
END_ACTION

ACTION ComToSPS:
(*Fehlermeldung auswerten und rangieren : Ist das Fehlerbit gesetzt, so wird die Fehlernummer ausgegeben.
  Liegt kein Fehler vor, so wird eine Null ausgegeben.*)	
 	IF stoerung 
	THEN  
		OUT_FEHLERNUMMER :=(PD_IN.PD_3_Status);
	END_IF
	
	IF NOT stoerung 
	THEN
		OUT_FEHLERNUMMER :=0;
	END_IF

//Setzten des Bits FU-Betriebbereit********************************************
	IF umrichter_bb 
	THEN 
		OUT_Status.NICHT_BEREIT := FALSE;
		ELSE
			OUT_Status.nicht_bereit :=TRUE;
	END_IF
	
	//Setzen des Bits FU-Störung********************************************
	IF stoerung 
		//AND NOT umrichter_bb
	THEN 
		OUT_STOERUNG := TRUE;
		ELSE 
			OUT_STOERUNG := FALSE;
	END_IF
	
	//Ausgabe ISt-Drehzahl***************************************************
	TEMP_IST_DREHZAHL_DINT :=INT_TO_DINT(WORD_TO_INT(PD_IN.PD_2_IST_DREHZAHL));
	DREHZAHL := DINT_TO_REAL(TEMP_IST_DREHZAHL_DINT);	
	
	IF inout_Visu.Para.Drehtausch
	THEN
		OUT_Status.ist_drehzahl := (DREHZAHL)*(-1);
	ELSE
		OUT_Status.ist_drehzahl := DREHZAHL;
	END_IF
	
	//Ausgabe IST-STROM***************************************************	
Out_Status.ist_strom:=WORD_TO_REAL(PD_IN.PD_5_IST_STROM);

////Ausgabe IST-Drehzahl***************************************************	
Out_Status.ist_strom:=WORD_TO_REAL(PD_IN.PD_4_IST_DREHMOMENT);

//Ausgabe Status Motoraktiv
Out_Status.antriebAktiv := ABS(OUT_Status.ist_drehzahl) > 1;

//Ausgabe Status Motor dreht mindestens 90% der Sollgeschwinidigkeit
Out_Status.ist_drehzahl_90 :=ABS( OUT_Status.ist_drehzahl) >= ABS(DREHZAHL * 0.9);
END_ACTION

ACTION Fehlerhandling:
//Fehler /Störung löschen*************************************************************************
	IF IN_QUITTIEREN 
	THEN 
		reset:= TRUE;
		ELSE 
			reset:= FALSE;
	END_IF
END_ACTION

ACTION Freigaben:
//Antrieb starten ,stoppen mit Rampe************************************************************
	IF start_stop
		OR Jog_pos
		OR Jog_neg
	THEN 
		freigabe_halt := TRUE;
	ELSE
		freigabe_halt := FALSE;
		PD_out.PD_2_solldrehzahl := DWORD_TO_WORD (REAL_TO_DWORD (0));
	END_IF


//Reglersperre setzen**************************************************************************
	reglersperre:=NOT IN_Reglersperre;
	freigabe_stop:= NOT IN_Reglersperre AND (freigabe_halt OR motor_dreht);
	
	freigabe_stop := NOT IN_Reglersperre;		// Muss nochmal genauer angeschaut werden - Andreas Funk
	freigabe_halt := NOT IN_Reglersperre;		// Muss nochmal genauer angeschaut werden - Andreas Funk
	
	IF IN_Reglersperre THEN
		inout_Visu.plus_start := FALSE;
		inout_Visu.minus_stop := FALSE;
		inout_steuern.vor := FALSE;
		inout_steuern.zur := FALSE;
	END_IF
END_ACTION

ACTION Handbetrieb:
// Wenn Maximaler Override nicht parametriert dann max Override 100%
IF inout_visu.Para.Max_Override_Hand = 0
THEN
	inout_visu.Para.Max_Override_Hand :=100;
END_IF

//===========================================
//###	Handgeschwinidgkeit schreiben	###
//===========================================

//---Override limitieren---
IF inout_visu.override > inout_visu.Para.Max_Override_Hand
THEN
	inout_visu.override := inout_visu.Para.Max_Override_Hand;
END_IF

//---Geschwinidgkeit berechnen

TEMP_DREHZAHL_SOLL:= REAL_TO_WORD(inout_Visu.Para.Speed_Hand / 10 * inout_visu.override);

inout_Visu.istdrehzahl:=INT_TO_REAL(WORD_TO_INT(PD_in.PD_2_IST_DREHZAHL))/10.0;

//---PD-Sollgeschwinidgkeit beschreiben---
IF in_Steuerstatus.hand
THEN
	IF  (inout_Visu.betriebsart = 1 AND inout_visu.plus_start AND NOT inout_Visu.Para.Drehtausch)
		OR (inout_Visu.betriebsart = 1 AND inout_visu.minus_stop AND inout_Visu.Para.Drehtausch)
		OR  (inout_Visu.betriebsart = 2 AND NOT inout_Visu.Para.Drehtausch)
		OR 	(inout_Visu.betriebsart = 4 AND inout_Visu.Para.Drehtausch)
	THEN
		PD_OUT.PD_2_Solldrehzahl:= TEMP_DREHZAHL_SOLL; 
	ELSIF
		(inout_Visu.betriebsart = 1 AND inout_visu.minus_stop AND NOT inout_Visu.Para.Drehtausch)
		OR (inout_Visu.betriebsart = 1 AND inout_visu.plus_start AND inout_Visu.Para.Drehtausch)
		OR  ((inout_Visu.betriebsart = 2 AND inout_Visu.Para.Drehtausch)
		OR 	(inout_Visu.betriebsart = 4 AND NOT inout_Visu.Para.Drehtausch))
	THEN	
		PD_OUT.PD_2_Solldrehzahl:= TEMP_DREHZAHL_SOLL*-1; 
	END_IF
	
END_IF

IF in_Steuerstatus.hand
THEN	

CASE inout_Visu.betriebsart OF 
0: // 
 hm_hand_vor	:= FALSE;
 hm_hand_zur	:= FALSE;
	
1:	//===========================================
	//###		Tippen		###
	//===========================================	
// ohne Drehrichtungstausch
IF NOT inout_Visu.Para.Drehtausch
THEN	
	IF inout_Visu.plus_start
	THEN
 		jog_pos:=TRUE;
		jog_neg:=FALSE;
		start_stop :=TRUE;
	ELSIF inout_Visu.minus_stop
	THEN
		jog_pos:=FALSE;
		jog_neg:=TRUE;
		start_stop :=TRUE;
	ELSE
		jog_pos:=FALSE;
		jog_neg:=FALSE;
		start_stop :=FALSE;
	END_IF
// mit Drehrichtungstausch	
ELSIF inout_Visu.Para.Drehtausch
THEN
	IF inout_Visu.plus_start
	THEN
 		jog_pos:=FALSE;
		jog_neg:=TRUE;
	ELSIF inout_Visu.minus_stop
	THEN
		jog_pos:=TRUE;
		jog_neg:=FALSE;
	ELSE
		jog_pos:=FALSE;
		jog_neg:=FALSE;
	END_IF
END_IF

2:	//===========================================
	//###		Kontinuierlich vorfahren	###
	//===========================================
	
IF inout_Visu.plus_start
THEN
		hm_hand_vor:=TRUE;
		inout_Visu.plus_start 	:= FALSE;
		
ELSIF inout_Visu.minus_stop
THEN
		hm_hand_vor			:= FALSE;
		inout_Visu.minus_stop 	:= FALSE;
		
END_IF		


start_Stop := hm_hand_vor;
4:	//===========================================
	//###		Kontinuierlich zurückfahren	###
	//===========================================
	
IF inout_Visu.plus_start
THEN
		hm_hand_zur:=TRUE;
		inout_Visu.plus_start 	:= FALSE;
		
ELSIF inout_Visu.minus_stop
THEN
		hm_hand_zur				:= FALSE;
		inout_Visu.minus_stop 	:= FALSE;
END_IF		
start_Stop := hm_hand_zur;


END_CASE


END_IF
		
IF inout_Visu.minus_stop
THEN
	inout_Visu.plus_start :=FALSE;
END_IF

IF inout_Visu.plus_start
THEN
	inout_Visu.minus_stop :=FALSE;
END_IF
END_ACTION

ACTION Rampen:
//************Vorgabe Soll-Rampe***************************************************************************
//---Defaultwerte setzen falls Beschleunigung nicht parametriert ist

//Beschleunigungsrampe
IF inout_visu.Para.Beschleunigung = 0
THEN
	inout_visu.Para.Beschleunigung := 500;
END_IF

//Verzögerungsrampe
IF inout_visu.Para.Verzoegerung = 0
THEN
	inout_visu.Para.Verzoegerung := 500;	
END_IF

//---Rampen beschreiben
PD_out.PD_3_Sollbeschleunigung 	:=REAL_TO_WORD(inout_visu.Para.Beschleunigung);
PD_out.PD_4_Sollverzoegerung 	:=REAL_TO_WORD(inout_visu.Para.Verzoegerung);
END_ACTION

ACTION Read_Statuswort:
//Statuswort auslesen*****************************************************************************************
	umrichter_bb		:= BIT_OF_dWORD(in:= PD_IN.PD_1_STATUSWORT, N:= 0);
	STO_inaktiv 		:= BIT_OF_dWORD(in:= PD_IN.PD_1_Statuswort, N:= 1);
	endstufe_freigegeben:= BIT_OF_DWORD(in:= PD_IN.PD_1_Statuswort, N:= 2);
	bremse_geoeffnet	:= BIT_OF_DWORD(in:= PD_IN.PD_1_Statuswort, N:= 3);
	motor_dreht			:= BIT_OF_DWORD(in:= PD_IN.PD_1_Statuswort, N:= 4);
	stoerung			:= BIT_OF_DWORD(in:= PD_IN.PD_1_Statuswort, N:= 8); // War vorher bit 5
END_ACTION

ACTION Status_CoE:
//300;Lese Parameter aus FU...
aktuellLesen:= CoE_ReadAndWrite.I_bStartRead
				AND NOT CoE_ReadAndWrite.I_bStartWriteFromCSV
				AND CoE_ReadAndWrite.Q_bBusy 
				AND NOT CoE_ReadAndWrite.Q_bError
				AND NOT CoE_ReadAndWrite.Q_bCSVDone
				AND NOT CoE_ReadAndWrite.Q_bWriteDone
				AND keinTimerAktiv;
	
//301;Lese Parameter aus FU erfolgreich

LesenErfolgreich:= NOT CoE_ReadAndWrite.I_bStartRead
				AND NOT CoE_ReadAndWrite.I_bStartWriteFromCSV
				AND NOT CoE_ReadAndWrite.Q_bBusy 
				AND NOT CoE_ReadAndWrite.Q_bError
				AND CoE_ReadAndWrite.Q_bCSVDone
				AND NOT CoE_ReadAndWrite.Q_bWriteDone
				AND keinTimerAktiv;
				
//302;Lese Parameter aus FU fehlgeschlagen

LesenFehlgeschlagen:=  CoE_ReadAndWrite.I_bStartRead
				AND NOT CoE_ReadAndWrite.I_bStartWriteFromCSV
				AND NOT CoE_ReadAndWrite.Q_bBusy 
				AND  CoE_ReadAndWrite.Q_bError
				AND NOT CoE_ReadAndWrite.Q_bCSVDone
				AND NOT CoE_ReadAndWrite.Q_bWriteDone
				AND keinTimerAktiv;
				
//306;Schreibe Parameter in FU...

aktuellSchreiben:= NOT CoE_ReadAndWrite.I_bStartRead
				AND CoE_ReadAndWrite.I_bStartWriteFromCSV
				AND CoE_ReadAndWrite.Q_bBusy 
				AND NOT CoE_ReadAndWrite.Q_bError
				AND NOT CoE_ReadAndWrite.Q_bCSVDone
				AND NOT CoE_ReadAndWrite.Q_bWriteDone
				AND keinTimerAktiv;

//307;Schreibe Parameter in FU erfolgreich

SchreibenErfolgreich:= NOT CoE_ReadAndWrite.I_bStartRead
				AND NOT CoE_ReadAndWrite.I_bStartWriteFromCSV
				AND NOT CoE_ReadAndWrite.Q_bBusy 
				AND NOT CoE_ReadAndWrite.Q_bError
				AND NOT CoE_ReadAndWrite.Q_bCSVDone
				AND CoE_ReadAndWrite.Q_bWriteDone
				AND keinTimerAktiv;
				
//308;Schreibe Parameter in FU fehlgeschlagen

SchreibenFehlgeschlagen:= NOT CoE_ReadAndWrite.I_bStartRead
				AND CoE_ReadAndWrite.I_bStartWriteFromCSV
				AND NOT CoE_ReadAndWrite.Q_bBusy 
				AND  CoE_ReadAndWrite.Q_bError
				AND NOT CoE_ReadAndWrite.Q_bCSVDone
				AND NOT CoE_ReadAndWrite.Q_bWriteDone
				AND keinTimerAktiv;
END_ACTION

ACTION Write_Steuerwort:
//Steuerwort schreiben
	steuerbyte_1	:= BYTE_OF_BIT(
	B0:= freigabe_stop, 
	B1:= freigabe_halt , 
	B2:= FALSE, 
	B3:= FALSE, 
	B4:= jog_pos, 
	B5:= jog_neg, 
	B6:= FALSE, 
	B7:= start_stop);
	
	steuerbyte_2 :=BYTE_OF_BIT(
	B0:= reset , 
	B1:= FALSE, 
	B2:= FALSE, 
	B3:= FALSE, 
	B4:= TRUE, 
	B5:= NOT reglersperre, 
	B6:= reserve_14  , 
	B7:= reserve_15);
    PD_out.PD_1_Steuerwort :=WORD_OF_BYTE(B1:= steuerbyte_2 , B0:=steuerbyte_1 );
	
(* Steuerwort --------------------------------------------------------------------
	BIT 0: Reglersperre
	0 = Freigabe
	1 = Regler sperren, Bremse aktivieren
	--------------------------------------------------------------------------------
	BIT 1: Freigabe/Schnellstopp
	0 = Schnellstopp
	1 = Freigabe
	--------------------------------------------------------------------------------
	BIT 2: Freigabe/Halt
	0 = Halt an Integratorrampe oder Prozess-Rampe
	1 = Freigabe
	--------------------------------------------------------------------------------
	BIT 3: Reserviert (Reservierte Bits sind generell auf Null zu setzen!)
	--------------------------------------------------------------------------------
	BIT 4: Reserviert (Reservierte Bits sind generell auf Null zu setzen!)
	--------------------------------------------------------------------------------
	BIT 5: Reserviert (Reservierte Bits sind generell auf Null zu setzen!)
	--------------------------------------------------------------------------------
	BIT 6: Reset
	0 = nicht aktiv
	0 -> 1 = anstehende Störung zurücksetzen
	--------------------------------------------------------------------------------
	BIT 7: Reserviert (Reservierte Bits sind generell auf Null zu setzen!)
	--------------------------------------------------------------------------------
	BIT 8: Drehrichtung für Motorpoti
	0 = Drehrichtung RECHTS
	1 = Drehrichtung LINKS
	--------------------------------------------------------------------------------
	BIT 10 und 9: Motorpoti Hochlauf,Motorpoti Tieflauf
	0 0 = keine Änderung
	1 0 = ab
	0 1 = auf
	1 1 = keine Änderung
	--------------------------------------------------------------------------------
	BIT 12 und 11:Anwahl der internen Festsollwerte
	n11...n13 bzw. n21...n23
	0 0 = Drehzahl-Sollwert über Prozess-Ausgangsdatenwort 2
	0 1 = interner Sollwert n11 (n21)
	1 0 = interner Sollwert n12 (n22)
	1 1 = interner Sollwert n13 (n23)
	--------------------------------------------------------------------------------
	BIT 13: Festsollwert-Umschaltung
	0 = Festsollwerte des aktivn Parametersatzes über Bit 11/12 anwählbar
	1 = Festsollwerte des anderen Parametersatzes über Bit 11/12 anwählbar
	--------------------------------------------------------------------------------
	BIT 14: Reserviert (Reservierte Bits sind generell auf Null zu setzen!)
	--------------------------------------------------------------------------------
	BIT 15: Reserviert (Reservierte Bits sind generell auf Null zu setzen!*)
END_ACTION

END_FUNCTION_BLOCK

// ---- SRT_Allgemein/0010_Bausteine_mitDuts/POUs/FB_Belegt.TcPOU
FUNCTION_BLOCK FB_Belegt 
VAR_INPUT
	in_Sensor			:BOOL;	
	in_zeit_ein			:TIME;	(* Zeitverzögert EIN - Sensor entprellen *)
	in_zeit_aus			:TIME;	(* Zeitverzögert AUS - Sensor entprellen *)
END_VAR
VAR_OUTPUT
	Q 					:BOOL;	(* Belegtmeldung - Eingang entprellt *)
	Qin					:BOOL;	(* orginal Signal ohne Zeiten*)	
	nFlanke				:BOOL;	(* Wird true bei negativer Flanke*)
	pFlanke				:BOOL;	(* Wird true bei positiver Flanke*)
END_VAR
VAR
	ein					:ton;
	aus					:tof;
	
	rTrig_pFlanke		:R_Trig;
	fTrig_nFlanke		:F_Trig;
END_VAR

//Belegtmeldung verzögert ein
ein(IN:=in_Sensor,
	PT:=in_zeit_ein);
	
//Belegtmeldung verzögert aus
aus(IN:=ein.Q,
	PT:=in_zeit_aus);

//Positive Flanke
rTrig_pFlanke(CLK:=ein.Q);

//Negative Flanke
fTrig_nFlanke(CLK:=aus.Q);

//Ausgänge zuweisen	
Q :=aus.Q;

pFlanke		:=rTrig_pFlanke.Q;
nFlanke		:=fTrig_nFlanke.Q;
Qin			:=in_Sensor;

END_FUNCTION_BLOCK

// ---- SRT_Allgemein/0010_Bausteine_mitDuts/POUs/FB_Ventil_V2.TcPOU
FUNCTION_BLOCK FB_Ventil_V2
(*
	Ansteuerungsbaustein zum Steuern und Überwachen von Ventilen und den dazugehörigen Sensoren
	(abgeleitet vom Siemens Baustein "Allg-Ventilbaustein" Stand 20.01.20)
	Autor O.E.
	Erstellt 20.01.20
	Version 1.0 
	
	Autor A.F.
	Erstellt 25.11.25
	Version 2.0
		- Vereinfachung / Verkürzung vom Programm
		- Methodenaufruf für Zylinder Ein bzw Aussteuern 
*)
VAR_INPUT
	in_endlage_vor	:BOOL;	(*1=Endlage vorne ist angefahren*)
	in_endlage_zur	:BOOL;	(*1=Endlage zurück ist angefahren*)
	in_hand			:BOOL;	(*1=Handbetrieb*)
	in_auto			:BOOL;	(*1=Automatikbetrieb*)
	in_quit			:BOOL;	(*		*)
END_VAR

VAR_OUTPUT
	out_vor				:BOOL;				(*Ausgang vorfahren*)
	out_zur				:BOOL;				(*Ausgang zurückfahren*)
	out_stoerung_vor	:BOOL;				(*Störung*)
	out_stoerung_zur	:BOOL;				(*Störung*)
	out_stoerung_vorzur	:BOOL;				(*Störung*)
	out_vor_visu		:BOOL;				(*Endlagen direkt für die Visu weitergeleitet*)
	out_zur_visu		:BOOL;				(*Endlagen direkt für die Visu weitergeleitet*)
END_VAR

VAR_IN_OUT
	inout_ansteuerung	:DUT_Ventil_sps;
	inout_visu			:DUT_Ventil_VISU;
END_VAR

VAR
	temp_zeit_vor				:TIME;
	temp_zeit_zur				:TIME;
	temp_zeit_entprellen_vor	:TIME;
	temp_zeit_entprellen_zur	:TIME;
	temp_end_vor				:BOOL;
	temp_end_zur				:BOOL;
	temp_stoer_vor				:BOOL;
	temp_stoer_zur				:BOOL;
	temp_stoer_vor_zur			:BOOL;	
END_VAR

VAR	
	verzoegerung_vor			:TON;	
	verzoegerung_zur			:TON;		
	ueberwachung_vor			:TON;		
	ueberwachung_zur			:TON;	
	fl_hm_vor					:R_trig;	
	fl_hm_zur					:R_trig;	

	hm_vor						:BOOL;	
	hm_zur						:BOOL;	
	hm_timer_reset				:BOOL;	
	hm_timer_reset_2			:BOOL;	
END_VAR

(************************************************************************************************************************************************************)
(*	SIGNALE IN 
		in_endlage_vor		--- 1 = Endlage vorne ist angefahren
		in_endlage_zur		--- 1 = Endlage zurück ist angefahren
		in_hand				--- Handbetrieb
		in_auto				--- Automatikbetrieb
		in_quit				--- Störungs Reset
						
	SIGNALE OUT 
		out_vor				--- Ausgang vorfahren
		out_zur				--- Ausgang zurückfahren
		out_stoerung		--- Störung
	
	SIGNALE INOUT - SPS
		in_auto_vor			--- Startsignal vorfahren (bleibt gespeichert)
		in_auto_zur			--- Startsignal zurückfahren (bleibt gespeichert)
		in_aus				--- intern gespeicherte Startsignale löschen
		in_freigabe_vor		--- 1 = vorfahren freigegeben
		in_freigabe_zur		--- 1 = zurückfahren freigegeben
		
		out_ist_vor			--- steht in Endlage vor und kein Fehler
		out_ist_zur			---	steht in Endlage zur und kein Fehler
	
	SIGNALE INOUT - VISU
		hand_vor			--- Hand vorfahren
		hand_zur			--- Hand zurückfahren
		reset				--- ntern gespeicherte Startsignale löschen
		service				--- 1 = ALLE Überwachungen deaktiviert
		status				--- 0=??? 1=vor 2=ist vor 3=fehler vor 4=zur 5=ist zur 6=Fehler zur 7=Fehler vor zur
		para				--- Parameter Struktur
			ueberwachung_vor_aktiv	--- 0 = Endlagenüberwachung vor deaktiviert
			ueberwachung_zur_aktiv	--- 0 = Endlagenüberwachung zurück deaktiviert
			ausgang_vor_halten		--- 1 = Ausgang immer Ein, sonst 0 in Endlage/1 nicht in Endlage
			ausgang_zur_halten		--- 1 = Ausgang immer Ein, sonst 0 in Endlage/1 nicht in Endlage
			entprellen_vor_aktiv	--- 0 = Endlage sofort überwachen wenn einmal erreicht
			entprellen_zur_aktiv	--  0 = Endlage sofort überwachen wenn einmal erreicht
			ueberwachungszeit_vor	--- Überwachungszeit in ms (0-30000ms)
			ueberwachungszeit_zur	--- Überwachungszeit in ms (0-30000ms)
			entprellungszeit_vor	--- Entprellungszeit in ms (0-10000ms)
			entprellungszeit_zur	--- Entprellungszeit in ms (0-10000ms)																					*)
(************************************************************************************************************************************************************)


(****** Zeitvorgabe prüfen **********************************************************************************************************************************)
(* Überwachung vor -> 0-300000ms  *)
	temp_zeit_vor:=inout_visu.para.ueberwachungszeit_vor;
	temp_zeit_vor := LIMIT(T#0MS, inout_visu.para.ueberwachungszeit_vor, T#30000MS);
(* Überwachung zurück -> 0-300000ms *)
	temp_zeit_zur:=inout_visu.para.ueberwachungszeit_zur;
	temp_zeit_zur := LIMIT(T#0MS, inout_visu.para.ueberwachungszeit_zur, T#30000MS);
(* Entprellen vor -> 0-10000s *)
	temp_zeit_entprellen_vor:=inout_visu.para.entprellungszeit_vor;
	temp_zeit_entprellen_vor := LIMIT(T#0MS, inout_visu.para.entprellungszeit_vor, T#10000MS);
(* Entprellen zurück -> 0-10000ms *)
	temp_zeit_entprellen_zur:=inout_visu.para.entprellungszeit_zur;
	temp_zeit_entprellen_zur := LIMIT(T#0MS, inout_visu.para.entprellungszeit_zur, T#10000MS);
	
(****** Endlage vor **********************************************************************************************************************************)
	verzoegerung_vor(IN:= in_endlage_vor
						AND NOT in_endlage_zur
						AND NOT hm_zur
						AND hm_timer_reset,
						pt:= temp_zeit_entprellen_vor);
	temp_end_vor:=((verzoegerung_vor.Q
					AND NOT inout_visu.service)
					OR (hm_vor
						AND inout_visu.service));
(****** Endlage zur **********************************************************************************************************************************)
	verzoegerung_zur(IN:= in_endlage_zur
						AND NOT in_endlage_vor
						AND NOT hm_vor
						AND hm_timer_reset,
						pt:= temp_zeit_entprellen_zur);
	temp_end_zur:=((verzoegerung_zur.Q
					AND NOT inout_visu.service)
					OR (hm_zur
						AND inout_visu.service));
(****** Start vor **********************************************************************************************************************************)
	IF ((in_auto
			AND inout_ansteuerung.in_auto_vor)
		OR (in_hand
			AND inout_visu.hand_vor))
		AND inout_ansteuerung.in_freigabe_vor
		AND NOT inout_ansteuerung.in_aus
	THEN
		hm_vor:=TRUE;
	END_IF
	
	IF (in_auto
			AND inout_ansteuerung.in_auto_zur)
		OR (in_hand
			AND inout_visu.hand_zur)
		OR inout_visu.reset
		OR inout_ansteuerung.in_aus
	THEN
		hm_vor:=FALSE;
	END_IF
	
	out_vor:=hm_vor
				AND inout_ansteuerung.in_freigabe_vor
				AND (NOT temp_end_vor
						OR inout_visu.para.ausgang_vor_halten);

(****** Start zur **********************************************************************************************************************************)
	IF ((in_auto
			AND inout_ansteuerung.in_auto_zur)
		OR (in_hand
			AND inout_visu.hand_zur))
		AND inout_ansteuerung.in_freigabe_zur
		AND NOT inout_ansteuerung.in_aus
	THEN
		hm_zur:=TRUE;
	END_IF

	IF (in_auto
			AND inout_ansteuerung.in_auto_vor)
		OR (in_hand
			AND inout_visu.hand_vor)
		OR inout_visu.reset
		OR inout_ansteuerung.in_aus
	THEN
		hm_zur:=FALSE;
	END_IF
	
	out_zur:=hm_zur
				AND inout_ansteuerung.in_freigabe_zur
				AND (NOT temp_end_zur
						OR inout_visu.para.ausgang_zur_halten);

(****** Flankenbildung bei vor und zurück *************************************************************************************************************)
(*wird benötigt damit der Timer bei direkten umschalten neu startet*) 
	fl_hm_vor(CLK:=hm_vor);
	fl_hm_zur(CLK:=hm_zur);
	
	hm_timer_reset_2:=fl_hm_vor.Q
					OR fl_hm_zur.Q
					OR ( NOT hm_vor
							AND NOT hm_zur)
					OR NOT inout_visu.para.ueberwachung_vor_aktiv	
					OR NOT inout_visu.para.ueberwachung_zur_aktiv	
					OR (out_stoerung_vorzur
						AND (temp_end_vor
								OR temp_end_zur))
					OR (hm_vor
						AND temp_end_vor)			
					OR (hm_zur
						AND temp_end_zur);			
	
(****** Zeitüberwachung Vor starten  *************************************************************************************************************)
	ueberwachung_vor(IN:=inout_visu.para.ueberwachung_vor_aktiv
							AND hm_vor
							AND NOT hm_timer_reset_2,
						pt:=temp_zeit_vor);
		
(****** Zeitüberwachung Zur starten  *************************************************************************************************************)
	ueberwachung_zur(IN:=inout_visu.para.ueberwachung_zur_aktiv
							AND hm_zur
							AND NOT hm_timer_reset_2,
						pt:=temp_zeit_zur);
		
(****** Störung - Zeitüberwachung Vor abgelaufen = Fehler *****************************************************************************************)
	temp_stoer_vor:=ueberwachung_vor.Q
					AND NOT temp_end_vor;
				
(****** Störung - Zeitüberwachung Zurück abgelaufen = Fehler **************************************************************************************)
	temp_stoer_zur:=ueberwachung_zur.Q
					AND NOT temp_end_zur;
	
(****** Störung - Beide Endlagen belegt = Fehler ***************************************************************************************************)
	temp_stoer_vor_zur:=temp_stoer_vor
						AND temp_stoer_zur;

(****** Störung - Ausgabe - STATUS auf 0 ************************************************************************************************************)
	IF in_quit
	THEN
		hm_timer_reset_2		:=FALSE;
		inout_visu.status		:=0;
	 	out_stoerung_vorzur		:=FALSE;
		out_Stoerung_vor		:=FALSE;
		out_Stoerung_zur		:=FALSE;
	END_IF						

	IF temp_stoer_vor
		AND NOT temp_stoer_vor_zur
	THEN
	 	out_stoerung_vor:=TRUE;
	END_IF						

	IF temp_stoer_zur
		AND NOT temp_stoer_vor_zur
	THEN
	 	out_stoerung_zur:=TRUE;
	END_IF						

	IF temp_stoer_vor_zur
	THEN
	 	out_stoerung_vorzur:=TRUE;
	END_IF						

	
(****** steht in Endlage vor und kein Fehler ********************************************************************************************************)
	inout_ansteuerung.out_ist_vor:= NOT out_stoerung_vorzur
									AND temp_end_vor;

(****** steht in Endlage zurück und kein Fehler *****************************************************************************************************)
	inout_ansteuerung.out_ist_zur:= NOT out_stoerung_vorzur
									AND temp_end_zur;
									
(***** Status ****************************************************************************************************************************************)
	(* 1=vor *)							
	IF hm_vor
		AND NOT temp_end_vor
		AND NOT temp_stoer_zur
		AND NOT temp_stoer_vor_zur
	THEN
		inout_visu.status:=1;									
	END_IF									
	(* 2=ist vor *)							
	IF (temp_end_vor
		OR (NOT inout_visu.para.ueberwachung_vor_aktiv
				AND hm_vor))
		AND NOT temp_end_zur
		AND NOT temp_stoer_zur
		AND NOT temp_stoer_vor_zur
	THEN
		inout_visu.status:=2;									
	END_IF															
	(* 3=Fehler vor	*)							
	IF temp_stoer_vor
	THEN
		inout_visu.status:=3;
	END_IF
	
